# B&R Automation Studio project MIG1
Automation Studio 4.12.7.113 SP; technology packages: Acp10Arnc0 1.0.0

## Configuration X20CP0484

CPU X20CP0484-1, AutomationRuntime E4.53, Build 4.1.2, Vc V4.52.0

### Task classes (Cpu.sw)
```
Cyclic#1 (cycle 1000 us, tolerance 10000 us):
  ESAB <- ESAB.prg
  LincolnPS <- LincolnPS.prg
  UDP_Client <- UDP_Client.prg
  TML_srv <- TML_srv.prg
Cyclic#2 (cycle 4000 us, tolerance 40000 us):
  MainProc <- MainProc.prg
Cyclic#3 (cycle 8000 us, tolerance 48000 us):
  Master <- Master.prg
Cyclic#4 (cycle 100000 us, tolerance 100000 us):
  HMI <- HMI.prg
Cyclic#8 (cycle 10000 us, tolerance 30000000 us):
  Program <- Program.prg [disabled]
  UDP <- UDP.prg [disabled]
  TcpCam <- TcpCam.prg [disabled]
VcDataObjects: Visu <- Visu.dob
Binaries: vcpfgen, vcnet, udbdef, vcrt, vcctext, vctcal, vccslider, Visu03, vcfile, vcgclass, vcpdsw, vccshape, arial, vccbmp, vcmgr, vcchspot, vcdsloc, vcfntttf, Visu02, vccovl, vcshared, arialbd, vcalarm, vcpdvnc, vccbtn, vcbclass, vcdsint, vccpwd, TCData, vccnum, Visu01, vccstr, vccpopup, vccddbox, vccdt, vccline, vcclbox, visvc, verabd, arialbi, vcpkat, vcctrend, iomap, asfw, Role, ashwac, sysconf, ashwd, User, arconfig
Libraries: AsXml, AsUDP, runtime, ETHERNET, standard, dvframe, asstring, AsTCP, AsHydCon, sys_lib, FileUser, FileIO, brsystem, LoopConR, DataObj, AsIOTime, XMLp_Lib, AsMbTCPS, AsMbTCP, vcresman, astime, visapi
```

### Hardware
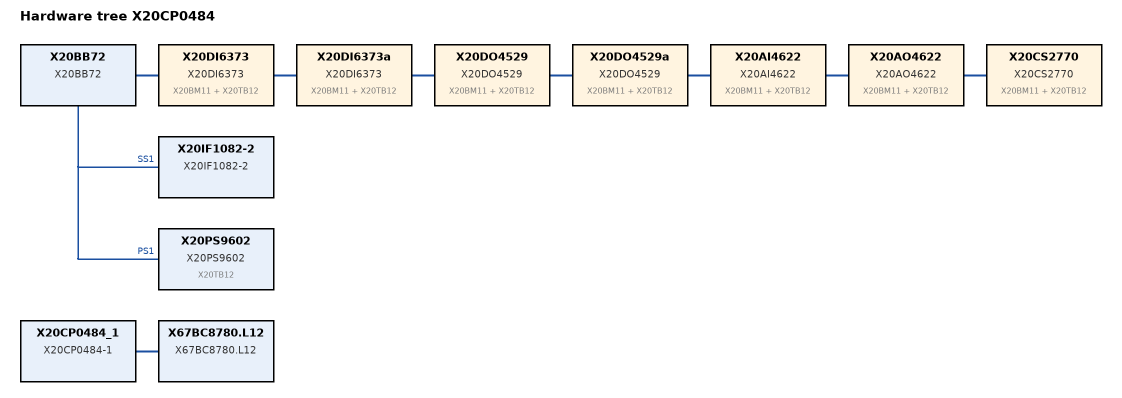
```
X20AI4622 : X20AI4622 v1.0.5.0  [SS1 -> X20TB12a.SS; SL -> X20BM11.SL1]
  Supervision = off
X20AO4622 : X20AO4622 v1.1.0.0  [SS1 -> X20TB12b.SS; SL -> X20BM11a.SL1]
  Supervision = off
X20BB72 : X20BB72 v1.2.0.0
  Connector IF1:
    ActivateIna = 0
  Connector IF6:
    CycleTime = 1000
X20BM11 : X20BM11 v1.1.0.0  [X2X1 -> X20BM11d.X2X2]
X20BM11a : X20BM11 v1.1.0.0  [X2X1 -> X20BM11.X2X2]
X20BM11b : X20BM11 v1.1.0.0  [X2X1 -> X20BB72.IF6]
X20BM11c : X20BM11 v1.1.0.0  [X2X1 -> X20BM11n.X2X2]
X20BM11d : X20BM11 v1.1.0.0  [X2X1 -> X20BM11c.X2X2]
X20BM11m : X20BM11 v1.1.0.0 (Disabled=true)  [X2X1 -> X20BM11a.X2X2]
X20BM11n : X20BM11 v1.1.0.0  [X2X1 -> X20BM11b.X2X2]
X20CP0484_1 : X20CP0484-1 v1.4.0.0
  Connector IF2:
    ActivateDevice = 1
  Connector IF3:
    DNAConfiguration = manual
  ConfigurationID = RemWeld_Config1
  PermanentPvSize = 2048
  RemanentGlobalPvSize = 128
  TimerDeviceType = EPLX2X
  TimerDevice = X20CP0484_1.IF3
  Cyclic1Duration = 1000
  Cyclic1Tolerance = 10000
  Cyclic2Duration = 4000
  Cyclic2Tolerance = 40000
  Cyclic3Duration = 8000
  Cyclic3Tolerance = 48000
  Cyclic4Duration = 100000
  Cyclic4Tolerance = 100000
  Cyclic5Duration = 200000
  Cyclic5Tolerance = 200000
  Cyclic6Duration = 500000
  Cyclic6Tolerance = 500000
  Cyclic7Duration = 1000000
  Cyclic7Tolerance = 1000000
  Cyclic8Duration = 10000
  Cyclic8Tolerance = 30000000
X20CS2770 : X20CS2770 v1.9.1.0 (Disabled=true)  [SS1 -> X20TB12n.SS; SL -> X20BM11m.SL1]
  Connector IF1 (Disabled=true)
  Connector IF2 (Disabled=true)
  Supervision = off
  CANdataFormat01 = UINT
  Baudrate02 = 250000
  CANdataFormat02 = UINT
X20DI6373 : X20DI6373 v1.0.1.0  [SS1 -> X20TB12c.SS; SL -> X20BM11b.SL1]
  Supervision = off
X20DI6373a : X20DI6373 v1.0.1.0  [SS1 -> X20TB12o.SS; SL -> X20BM11n.SL1]
  Supervision = off
X20DO4529 : X20DO4529 v1.2.0.0  [SS1 -> X20TB12d.SS; SL -> X20BM11c.SL1]
  Supervision = off
X20DO4529a : X20DO4529 v1.2.0.0  [SS1 -> X20TB12e.SS; SL -> X20BM11d.SL1]
  Supervision = off
X20IF1082-2 : X20IF1082-2 v1.14.0.0  [SS -> X20BB72.SS1]
  Connector IF1:
    EplNatSubnet = 192.168.102.0
X20PS9602 : X20PS9602 v1.1.0.0  [PS -> X20BB72.PS1; SS1 -> X20TB12.SS]
  Supervision = off
X20TB12 : X20TB12 v1.0.0.0
X20TB12a : X20TB12 v1.0.0.0
X20TB12b : X20TB12 v1.0.0.0
X20TB12c : X20TB12 v1.0.0.0
X20TB12d : X20TB12 v1.0.0.0
X20TB12e : X20TB12 v1.0.0.0
X20TB12n : X20TB12 v1.0.0.0 (Disabled=true)
X20TB12o : X20TB12 v1.0.0.0
X67BC8780.L12 : X67BC8780.L12 v2.14.0.0 (Disabled=true)  [PLK1 -> X20CP0484_1.IF3 [Cable Type=PowerlinkCable, Length=10, Version=1.0.0.3]]
  Connector IF1 (Disabled=true)
```

### Cpu.per - X20CP0484_1/Cpu.per
```iecst
VAR_CONFIG
	permMemInit AT %MX0; (* *)
	TravelSpeed AT %M4; (* *)
	OLD_MTR_POS AT %MD8; (* *)
	CurCalib AT %M72; (* *)
	permMem AT %M468; (* *)
	MachCfg AT %M1620; (* *)
END_VAR
```

### IoMap.iom - X20CP0484_1/IoMap.iom
```iecst
VAR_CONFIG
	::TML_mgr[0].hrdw[0].TXCountReadBack AT %IB."X20CS2770".TX01CountReadBack;
	::TML_mgr[0].hrdw[0].RXDataSize0 AT %IB."X20CS2770".RX01DataSize;
	::TML_mgr[0].hrdw[0].RXIdent0 AT %ID."X20CS2770".RX01Ident;
	::TML_mgr[0].hrdw[0].RXData0Word0[0] AT %IW."X20CS2770".RX01DataWord0;
	::TML_mgr[0].hrdw[0].RXData0Word0[1] AT %IW."X20CS2770".RX01DataWord1;
	::TML_mgr[0].hrdw[0].RXData0Word0[2] AT %IW."X20CS2770".RX01DataWord2;
	::TML_mgr[0].hrdw[0].RXData0Word0[3] AT %IW."X20CS2770".RX01DataWord3;
	::TML_mgr[0].hrdw[0].TXCount AT %QB."X20CS2770".TX01Count;
	::TML_mgr[0].hrdw[0].TXDataSize AT %QB."X20CS2770".TX01DataSize; (*Data length TX object *)
	::TML_mgr[0].hrdw[0].TXIdent AT %QD."X20CS2770".TX01Ident;
	::TML_mgr[0].hrdw[0].TXDataWord0[0] AT %QW."X20CS2770".TX01DataWord0;
	::TML_mgr[0].hrdw[0].TXDataWord0[1] AT %QW."X20CS2770".TX01DataWord1;
	::TML_mgr[0].hrdw[0].TXDataWord0[2] AT %QW."X20CS2770".TX01DataWord2;
	::TML_mgr[0].hrdw[0].TXDataWord0[3] AT %QW."X20CS2770".TX01DataWord3;
	::TML_mgr[0].hrdw[1].RXCount AT %IB."X20CS2770".RX02Count;
	::TML_mgr[0].hrdw[1].TXCountReadBack AT %IB."X20CS2770".TX02CountReadBack;
	::TML_mgr[0].hrdw[1].RXDataSize0 AT %IB."X20CS2770".RX02DataSize;
	::TML_mgr[0].hrdw[1].RXIdent0 AT %ID."X20CS2770".RX02Ident;
	::TML_mgr[0].hrdw[1].RXData0Word0[0] AT %IW."X20CS2770".RX02DataWord0;
	::TML_mgr[0].hrdw[1].RXData0Word0[1] AT %IW."X20CS2770".RX02DataWord1;
	::TML_mgr[0].hrdw[1].RXData0Word0[2] AT %IW."X20CS2770".RX02DataWord2;
	::TML_mgr[0].hrdw[1].RXData0Word0[3] AT %IW."X20CS2770".RX02DataWord3;
	::TML_mgr[0].hrdw[1].TXCount AT %QB."X20CS2770".TX02Count;
	::TML_mgr[0].hrdw[1].TXDataSize AT %QB."X20CS2770".TX02DataSize; (*Data length TX object *)
	::TML_mgr[0].hrdw[1].TXIdent AT %QD."X20CS2770".TX02Ident;
	::TML_mgr[0].hrdw[1].TXDataWord0[0] AT %QW."X20CS2770".TX02DataWord0;
	::TML_mgr[0].hrdw[1].TXDataWord0[1] AT %QW."X20CS2770".TX02DataWord1;
	::TML_mgr[0].hrdw[1].TXDataWord0[2] AT %QW."X20CS2770".TX02DataWord2;
	::TML_mgr[0].hrdw[1].TXDataWord0[3] AT %QW."X20CS2770".TX02DataWord3;
	::Main_IO.Inp[0] AT %IX."X20DI6373".DigitalInput01;
	::VoltCmd_Out AT %QW."X20AO4622".AnalogOutput02;
	::Main_IO.Inp[1] AT %IX."X20DI6373".DigitalInput02;
	::Main_IO.Inp[2] AT %IX."X20DI6373".DigitalInput03;
	::Main_IO.Inp[3] AT %IX."X20DI6373".DigitalInput04;
	::Main_IO.Inp[4] AT %IX."X20DI6373".DigitalInput05;
	::Main_IO.Inp[5] AT %IX."X20DI6373".DigitalInput06;
	::Main_IO.Inp[6] AT %IX."X20DI6373a".DigitalInput01;
	::Main_IO.Inp[7] AT %IX."X20DI6373a".DigitalInput02;
	::Main_IO.Inp[8] AT %IX."X20DI6373a".DigitalInput03;
	::Main_IO.Inp[9] AT %IX."X20DI6373a".DigitalInput04;
	::Main_IO.Inp[10] AT %IX."X20DI6373a".DigitalInput05;
	::Main_IO.Inp[11] AT %IX."X20DI6373a".DigitalInput06;
	::Main_IO.Out[0] AT %QX."X20DO4529".DigitalOutput01;
	::Main_IO.Out[1] AT %QX."X20DO4529".DigitalOutput02;
	::Main_IO.Out[2] AT %QX."X20DO4529".DigitalOutput03;
	::Main_IO.Out[3] AT %QX."X20DO4529".DigitalOutput04;
	::Main_IO.Out[4] AT %QX."X20DO4529a".DigitalOutput01;
	::Main_IO.Out[5] AT %QX."X20DO4529a".DigitalOutput02;
	::Main_IO.Out[6] AT %QX."X20DO4529a".DigitalOutput03;
	::Main_IO.Out[7] AT %QX."X20DO4529a".DigitalOutput04;
END_VAR
```

## Configuration X20CP1585S

CPU X20CP1585, AutomationRuntime J4.93, Build 4.1.2, Safety 1.10, Vc V4.73.2

### Hardware
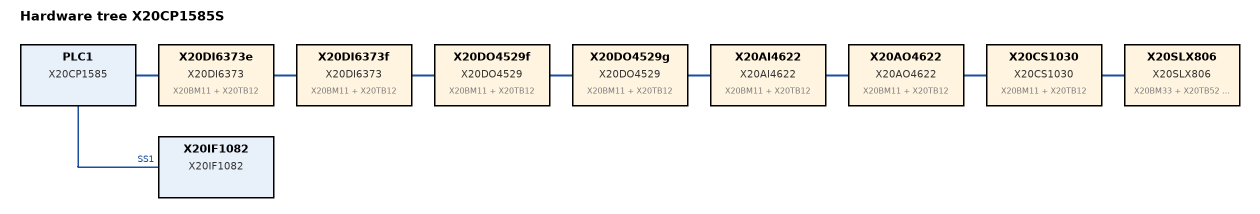
```
PLC1 : X20CP1585 v1.10.0.0
  Connector IF2:
    ActivateDevice = 1
    Mode = Manual
    InternetAddress = 192.168.10.123
    SubnetMask = 255.255.255.0
    Vnc1
    VncVcObjectName1 = Visu
    VncKeyMappingFile1 = VC\PS2-Keyboard.dis
    VncAuthentication1 = 1
    VncPasswordViewControl1 = c
    VncMaxConnections1 = 3
    VncRefreshRate1 = 100
    VncTitle1 = MIG
    Vnc2
    VncVcObjectName2 = Visu1
    VncKeyMappingFile2 = VC\PS2-Keyboard1.dis
    VncAuthentication2 = 1
    VncPasswordViewControl2 = c
    VncPortNumber2 = 5901
    VncRefreshRate2 = 200
  Connector IF3:
    ActivatePowerlink = 0
    DNAConfiguration = manual
    CycleTime = 800
    EplNatSubnet = 192.168.102.0
    HostName = pwl
    InternetAddress = 192.168.11.123
    SubnetMask = 255.255.255.0
    InaNodeNumber = 1
  Connector IF6:
    CycleTime = 800
  ConfigurationID = MIG-26July21
  UserPartitionSize = 256
  UserRamSize = 770048
  PermanentPvSize = 96000
  RemanentGlobalPvSize = 15000
  VolatileGlobalPvSize = 3300000
  TimerDeviceType = EPLX2X
  TimerDevice = PLC1.IF3
  TaskClassIdleTime = 1600
  Cyclic1Duration = 800
  Cyclic1Tolerance = 8000
  Cyclic1Stack = 16000
  Cyclic2Duration = 2400
  Cyclic2Tolerance = 24000
  Cyclic2Stack = 65536
  Cyclic3Duration = 4800
  Cyclic3Tolerance = 24000
  Cyclic4Duration = 24000
  Cyclic4Tolerance = 48000
  Cyclic4Stack = 65536
  Cyclic5Duration = 102400
  Cyclic5Tolerance = 204800
  Cyclic6Duration = 409600
  Cyclic6Tolerance = 409600
  Cyclic7Duration = 20000000
  Cyclic7Tolerance = 20000000
  Cyclic8Duration = 8000
  Cyclic8Tolerance = 40000000
  FileDevice1
  FileDeviceName1 = XML
  FileDevicePath1 = F:\XML
  FileDevice2
  FileDeviceName2 = USB1
  FileDevicePath2 = IF4
  FileDevice3
  FileDeviceName3 = USB2
  FileDevicePath3 = IF5
  FileDevice4
  FileDeviceName4 = REPORTS
  FileDevicePath4 = F:\Reports
  FtpUser1
  FtpUsername1 = anonymous
  FtpUserPassword1 = ilVrWe+rnGADVB+XCj+0qQ/lTsJeu4vW1xfWuH+9Xv8=
  FtpUserSalt1 = NATz6vdL
  FTPAccessRight1 = 0
X20AI4622 : X20AI4622 v1.0.5.0  [SS1 -> X20TB12.SS; SL -> X20BM11.SL1]
  Supervision = off
X20AO4622 : X20AO4622 v1.1.0.0  [SS1 -> X20TB12a.SS; SL -> X20BM11a.SL1]
  Supervision = off
X20BM11 : X20BM11 v1.1.0.0  [X2X1 -> X20BM11p.X2X2]
X20BM11a : X20BM11 v1.1.0.0  [X2X1 -> X20BM11.X2X2]
X20BM11b : X20BM11 v1.1.0.0  [X2X1 -> X20BM11a.X2X2]
X20BM11m : X20BM11 v1.1.0.0  [X2X1 -> PLC1.IF6]
X20BM11n : X20BM11 v1.1.0.0  [X2X1 -> X20BM11m.X2X2]
X20BM11o : X20BM11 v1.1.0.0  [X2X1 -> X20BM11n.X2X2]
X20BM11p : X20BM11 v1.1.0.0  [X2X1 -> X20BM11o.X2X2]
X20BM33 : X20BM33 v1.1.0.0 (Disabled=true)  [X2X1 -> X20BM11b.X2X2]
X20CS1030 : X20CS1030 v1.4.2.0  [SS1 -> X20TB12b.SS; SL -> X20BM11b.SL1]
  Supervision = off
X20DI6373e : X20DI6373 v1.0.1.0  [SS1 -> X20TB12q.SS; SL -> X20BM11m.SL1]
  Supervision = off
X20DI6373f : X20DI6373 v1.0.1.0  [SS1 -> X20TB12r.SS; SL -> X20BM11n.SL1]
  Supervision = off
X20DO4529f : X20DO4529 v1.2.0.0  [SS1 -> X20TB12s.SS; SL -> X20BM11o.SL1]
  Supervision = off
X20DO4529g : X20DO4529 v1.2.0.0  [SS1 -> X20TB12t.SS; SL -> X20BM11p.SL1]
  Supervision = off
X20IF1082 : X20IF1082 v1.6.0.0 (Disabled=true)  [SS -> PLC1.SS1]
  Connector IF1 (Disabled=true)
    ActivatePowerlink = 0
    DNAConfiguration = manual
    InternetAddress = 192.168.1.123
    SubnetMask = 255.255.255.0
X20SLX806 : X20SLX806 v1.10.12.1 (Disabled=true)  [SS1 -> X20TB52.SS; SS2 -> X20TB52a.SS; SL -> X20BM33.SL1]
  Supervision = off
  SafeProject = SafeLOGIC-1
  SafeDesigner = 4.2.5.4
X20TB12 : X20TB12 v1.0.0.0
X20TB12a : X20TB12 v1.0.0.0
X20TB12b : X20TB12 v1.0.0.0
X20TB12q : X20TB12 v1.0.0.0
X20TB12r : X20TB12 v1.0.0.0
X20TB12s : X20TB12 v1.0.0.0
X20TB12t : X20TB12 v1.0.0.0
X20TB52 : X20TB52 v1.0.0.1 (Disabled=true)
X20TB52a : X20TB52 v1.0.0.1 (Disabled=true)
```

- Safety project (password-protected, skipped)

## Configuration X20CP1685S

CPU X20CP1685, AutomationRuntime J4.93, Build 4.1.2, Safety 1.10, Vc V4.73.2

### Hardware
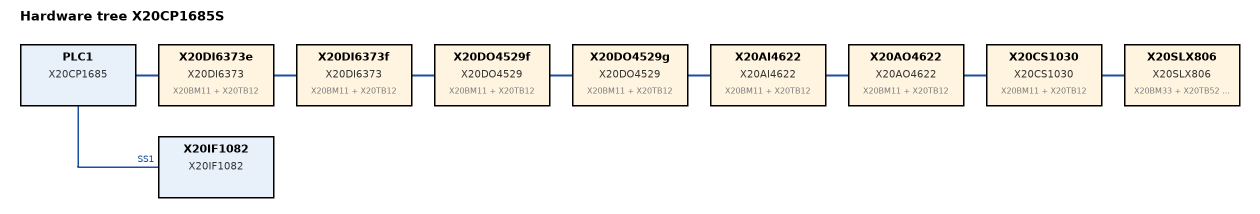
```
PLC1 : X20CP1685 v1.5.0.0
  Connector IF2:
    ActivateDevice = 1
    Mode = Manual
    InternetAddress = 192.168.10.123
    SubnetMask = 255.255.255.0
    Vnc1
    VncVcObjectName1 = Visu
    VncKeyMappingFile1 = VC\PS2-Keyboard.dis
    VncAuthentication1 = 1
    VncPasswordViewControl1 = c
    VncMaxConnections1 = 3
    VncRefreshRate1 = 100
    VncTitle1 = MIG
    Vnc2
    VncVcObjectName2 = Visu1
    VncKeyMappingFile2 = VC\PS2-Keyboard1.dis
    VncAuthentication2 = 1
    VncPasswordViewControl2 = c
    VncPortNumber2 = 5901
    VncRefreshRate2 = 200
  Connector IF3:
    ActivatePowerlink = 0
    DNAConfiguration = manual
    CycleTime = 800
    EplNatSubnet = 192.168.102.0
    HostName = pwl
    InternetAddress = 192.168.11.123
    SubnetMask = 255.255.255.0
    InaNodeNumber = 1
  Connector IF6:
    CycleTime = 800
  ConfigurationID = MIG-26July21
  UserPartitionSize = 256
  UserRamSize = 770048
  PermanentPvSize = 96000
  RemanentGlobalPvSize = 15000
  VolatileGlobalPvSize = 3300000
  TimerDeviceType = EPLX2X
  TimerDevice = PLC1.IF3
  TaskClassIdleTime = 1600
  Cyclic1Duration = 800
  Cyclic1Tolerance = 8000
  Cyclic1Stack = 16000
  Cyclic2Duration = 2400
  Cyclic2Tolerance = 24000
  Cyclic2Stack = 65536
  Cyclic3Duration = 4800
  Cyclic3Tolerance = 24000
  Cyclic4Duration = 24000
  Cyclic4Tolerance = 48000
  Cyclic4Stack = 65536
  Cyclic5Duration = 102400
  Cyclic5Tolerance = 204800
  Cyclic6Duration = 409600
  Cyclic6Tolerance = 409600
  Cyclic7Duration = 20000000
  Cyclic7Tolerance = 20000000
  Cyclic8Duration = 8000
  Cyclic8Tolerance = 40000000
  FileDevice1
  FileDeviceName1 = XML
  FileDevicePath1 = F:\XML
  FileDevice2
  FileDeviceName2 = USB1
  FileDevicePath2 = IF4
  FileDevice3
  FileDeviceName3 = USB2
  FileDevicePath3 = IF5
  FileDevice4
  FileDeviceName4 = REPORTS
  FileDevicePath4 = F:\Reports
  FtpUser1
  FtpUsername1 = anonymous
  FtpUserPassword1 = ilVrWe+rnGADVB+XCj+0qQ/lTsJeu4vW1xfWuH+9Xv8=
  FtpUserSalt1 = NATz6vdL
  FTPAccessRight1 = 0
X20AI4622 : X20AI4622 v1.0.5.0  [SS1 -> X20TB12.SS; SL -> X20BM11.SL1]
  Supervision = off
X20AO4622 : X20AO4622 v1.1.0.0  [SS1 -> X20TB12a.SS; SL -> X20BM11a.SL1]
  Supervision = off
X20BM11 : X20BM11 v1.1.0.0  [X2X1 -> X20BM11p.X2X2]
X20BM11a : X20BM11 v1.1.0.0  [X2X1 -> X20BM11.X2X2]
X20BM11b : X20BM11 v1.1.0.0  [X2X1 -> X20BM11a.X2X2]
X20BM11m : X20BM11 v1.1.0.0  [X2X1 -> PLC1.IF6]
X20BM11n : X20BM11 v1.1.0.0  [X2X1 -> X20BM11m.X2X2]
X20BM11o : X20BM11 v1.1.0.0  [X2X1 -> X20BM11n.X2X2]
X20BM11p : X20BM11 v1.1.0.0  [X2X1 -> X20BM11o.X2X2]
X20BM33 : X20BM33 v1.1.0.0 (Disabled=true)  [X2X1 -> X20BM11b.X2X2]
X20CS1030 : X20CS1030 v1.4.2.0  [SS1 -> X20TB12b.SS; SL -> X20BM11b.SL1]
  Supervision = off
X20DI6373e : X20DI6373 v1.0.1.0  [SS1 -> X20TB12q.SS; SL -> X20BM11m.SL1]
  Supervision = off
X20DI6373f : X20DI6373 v1.0.1.0  [SS1 -> X20TB12r.SS; SL -> X20BM11n.SL1]
  Supervision = off
X20DO4529f : X20DO4529 v1.2.0.0  [SS1 -> X20TB12s.SS; SL -> X20BM11o.SL1]
  Supervision = off
X20DO4529g : X20DO4529 v1.2.0.0  [SS1 -> X20TB12t.SS; SL -> X20BM11p.SL1]
  Supervision = off
X20IF1082 : X20IF1082 v1.6.0.0 (Disabled=true)  [SS -> PLC1.SS1]
  Connector IF1 (Disabled=true)
    ActivatePowerlink = 0
    DNAConfiguration = manual
    InternetAddress = 192.168.1.123
    SubnetMask = 255.255.255.0
X20SLX806 : X20SLX806 v1.10.12.1 (Disabled=true)  [SS1 -> X20TB52.SS; SS2 -> X20TB52a.SS; SL -> X20BM33.SL1]
  Supervision = off
  SafeProject = SafeLOGIC-1
  SafeDesigner = 4.2.5.4
X20TB12 : X20TB12 v1.0.0.0
X20TB12a : X20TB12 v1.0.0.0
X20TB12b : X20TB12 v1.0.0.0
X20TB12q : X20TB12 v1.0.0.0
X20TB12r : X20TB12 v1.0.0.0
X20TB12s : X20TB12 v1.0.0.0
X20TB12t : X20TB12 v1.0.0.0
X20TB52 : X20TB52 v1.0.0.1 (Disabled=true)
X20TB52a : X20TB52 v1.0.0.1 (Disabled=true)
```

### Cpu.per - PLC1/Cpu.per
```iecst
(********************************************************************
 * COPYRIGHT -- wsi
 ********************************************************************
 * File: Cpu.per
 * Author: wsi
 * Created: May 14, 2013
 ********************************************************************
 * Declaration of permanent variables
 ********************************************************************)
VAR_CONFIG
	permMemInit AT %MX0; (* *)
	TravelSpeed AT %M4; (* *)
	OLD_MTR_POS AT %MD8; (* *)
	CurCalib AT %M72; (* *)
	permMem AT %M468; (* *)
	MachCfg AT %M1620; (* *)
END_VAR
```

### IoMap.iom - PLC1/IoMap.iom
```iecst
(********************************************************************
 * COPYRIGHT -- wsi
 ********************************************************************
 * File: IoMap.iom
 * Author: wsi
 * Created: May 14, 2013
 ********************************************************************
 * IO mapping file
 ********************************************************************)
VAR_CONFIG
	::Main_IO.Inp[0] AT %IX."X20DI6373e".DigitalInput01;
	::Main_IO.Inp[1] AT %IX."X20DI6373e".DigitalInput02;
	::Main_IO.Inp[2] AT %IX."X20DI6373e".DigitalInput03;
	::Main_IO.Inp[3] AT %IX."X20DI6373e".DigitalInput04;
	::Main_IO.Inp[4] AT %IX."X20DI6373e".DigitalInput05;
	::Main_IO.Inp[5] AT %IX."X20DI6373e".DigitalInput06;
	::Main_IO.Inp[6] AT %IX."X20DI6373f".DigitalInput01;
	::Main_IO.Inp[7] AT %IX."X20DI6373f".DigitalInput02;
	::Main_IO.Inp[8] AT %IX."X20DI6373f".DigitalInput03;
	::Main_IO.Inp[9] AT %IX."X20DI6373f".DigitalInput04;
	::Main_IO.Inp[10] AT %IX."X20DI6373f".DigitalInput05;
	::Main_IO.Inp[11] AT %IX."X20DI6373f".DigitalInput06;
	::Main_IO.Out[0] AT %QX."X20DO4529f".DigitalOutput01;
	::Main_IO.Out[1] AT %QX."X20DO4529f".DigitalOutput02;
	::Main_IO.Out[2] AT %QX."X20DO4529f".DigitalOutput03;
	::Main_IO.Out[3] AT %QX."X20DO4529f".DigitalOutput04;
	::Main_IO.Out[4] AT %QX."X20DO4529g".DigitalOutput01;
	::Main_IO.Out[5] AT %QX."X20DO4529g".DigitalOutput02;
	::Main_IO.Out[6] AT %QX."X20DO4529g".DigitalOutput03;
	::Main_IO.Out[7] AT %QX."X20DO4529g".DigitalOutput04;
	::VoltCmd_Out AT %QW."X20AO4622".AnalogOutput02;
END_VAR
```

## Logical view

Binary libraries used (declarations not repeated): operator, runtime, astime, AsIecCon, AsUDP, standard, dvframe, asstring, AsTCP, AsHydCon 3.10.0, sys_lib, brsystem, LoopConR 4.10.0, DataObj, AsIOTime, AsMbTCPS, bglibas, AsXml, sprintf2, NcGlobal 3.13.1, Acp10man 3.13.1, Acp10par 3.13.1, AsMbTCP, AsSafety, FileIO, ETHERNET, visapi

### GlobalDef.h
```c
#include <bur/plctypes.h>

#ifndef _GLOBAL_DEF_H
#define _GLOBAL_DEF_H

#ifdef _DEFAULT_INCLUDES
#include <AsDefault.h>
#endif

#include <..\Lib\WSI_types.h>
#include <..\Lib\LoggerLib.h>

#include <..\Lib\arclink\arclink.h>

// "192.168.10.11"   	TML -> CAN conerter
// "192.168.10.2"   	Lincoln Power Supply
// "192.168.10.110"  	VNC - Pendant Screen
// "192.168.10.13" 		My Laptop

//#define SOFTWARE_VERSION    "MIG 09 June 2023V" // two new mode : 169 Carbon & 171 Stainless steel

//#define SOFTWARE_VERSION    "MIG 12 June 2023B" // two new mode : 169 Carbon & 171 Stainless steel

//#define SOFTWARE_VERSION    "MIG 14 June 2023H" // ta dziala przy tescie

//#define SOFTWARE_VERSION    "MIG 20 June 2023F" // FINAL GOOD VERSION req.: MIG 04 Nov 2022 new AHC Rel Move.m

//#define SOFTWARE_VERSION    "MIG 21 June 2023Y" //

//#define SOFTWARE_VERSION    "MIG 22 June 2023H" // Dobrze dziala - sprawdzona z Martin i David

//#define SOFTWARE_VERSION    "MIG 23 June 2023A" // Gas Solenoid in ArcLink

//#define SOFTWARE_VERSION    "MIG 9 Aug 2023C" // Nie dziala - przy stopie bez error WF jechal

//#define SOFTWARE_VERSION    "MIG 9 Aug 2023E"

//#define SOFTWARE_VERSION    "MIG 10 Aug 2023F" // DObra stabilna wersja
//#define SOFTWARE_VERSION    "MIG 11 Aug 2023F" // drobna poprawka w tekscie na ekranie

//#define SOFTWARE_VERSION    "MIG 23 Oct 2024A"  // weld report added

//#define SOFTWARE_VERSION    "MIG5 14 Nov 2024A"  // TVL indexing from trigger

//#define SOFTWARE_VERSION    "MIG 30 Jan 2025F"  // Ramp for amps in gauging , TVL indexing from trigger

//#define SOFTWARE_VERSION    "MIG 08 Aug 2025K"  // Gouging over current protection

//#define SOFTWARE_VERSION    "MIG 14 Aug 2025A"  // No Gouging over current protection & No repeat bead protection when gouging

//#define SOFTWARE_VERSION    "MIG 04 Sept 2025K"  // Report data display
//#define SOFTWARE_VERSION    "MIG 05 Sept 2025K"  // Report data display
#define SOFTWARE_VERSION    "MIG 26 Sept 2025F"  // bypass CheckIndxDone()

//////////////////////////////////////////
#define SERVO_NUM  6 // number of used servo

#define VISIBLE 	0
#define INVISIBLE 	1

#define MAX_PARAM_NUM 96

#define TravelSpeedAO_Indx 				0
#define ArcVoltsAO_Indx  				1
#define	WireFeedSpeedAO_Indx  			2
#define	AHCCurrentSPAO_Indx  			3
#define	AHCToleranceAO_Indx  			4
#define	OSCSpeedAO_Indx  				5

#define	Index_Dist_H_Indx  				6
#define Index_Dist_L_Indx				7

#define	Index_Jog_Speed_Indx  			8
#define	Index_Step_Speed_Indx  			9

#define	TVL_Jog_Speed_Indx  			10
#define WF_Jog_Speed_Indx  				11

#define	Index_PreDlyTime_Indx  			12
#define	Index_PostDlyTime_Indx  		13

////
#define	OSC_AmplitAO_Indx  				14
#define	OSC_DwellInAO_Indx  			15
#define	OSC_DwellOutAO_Indx  			16
#define	OSC_JogSpeedAO_Indx  			17
#define	OSC_StepDistAO_Indx  			18

/////
#define	AHC_JogSpeedAO_Indx  			19
#define AHC_Response_Indx  				20
#define AHC_Integrator_Indx  			21

////////////
#define TVL_Calibr_Vel_Low				25
#define TVL_Calibr_Vel_High				26
#define TVL_Calibr_Dist					27
////////////
#define WF_Calibr_Vel_Low				30
#define WF_Calibr_Vel_High				31
#define WF_Calibr_Time					32

/////// Ramps
#define TVL_Ramp						50
#define TVL_Return_Speed				51

#define WF_Ramp							52
#define TVL_Skip_Speed					53

////  GAS

#define GAS_PrePurge					54
#define GAS_PostPurge					55

////  Weld Mode

#define StanBy_Time						56
#define Weld_Pinch						57
#define Weld_Trim						58
#define Weld_UltimArc					59

#define AMPS_Calibr_Low					60
#define AMPS_Calibr_High				61

#define BURN_BACK_Tm					62

#define WF_SlowSpeed					63

#define AHC_Retrack_Dist  				64

#define GOUG_Volts  				    65
#define GOUG_Amps 				    	66

#define ARC_Start_Tmo					67
#define ARC_NotActive_Level				68

#define OSC_OFF_Tm						69

#define GOUG_Amps_Init 				    70
#define GOUG_Amps_Ramp 				    71

#define GOUG_Amps_Limit 				72
#define GOUG_Amps_Limit_Tm 				73

#define Wire_Dim 						74

#define	LastPermMem_Indx  				75

/////////////////////////////////////////////////
#define CALIBR_WF_Indx					0
#define CALIBR_AMPS_Indx				1
#define CALIBR_TVL_Indx					2

///////////////////////
#define WF_Calibr_Indx			0   // speed
#define AMPS_Calibr_Indx		1   // Amp feedback
#define TVL_Calibr_Indx			2   // speed

#define Index_Calibr_Indx		3   // distance
#define OSC_Calibr_Indx			4	// distance
#define ArcVolts_Calibr_Indx	5   // Volts to Power Supply

///////////////////////////
#define mm2inch 0.03936996
#define in_min_2_mm_s 25.4/60.0
#define in_2_mm 25.4

/////////   IO mapping
// Inputs

#define ESTOP_status 5

#define STOP_RST_BTN_LOC 6
#define STOP_RST_BTN 7

#define JOG1_BTN 9
#define JOG2_BTN 10

#define RESET_BTN_LOC 11

//outputs
#define ENABLE_out 3
#define RESET_ESR_Btn_out 4

typedef struct HEAD_typ
{
	plcbit Remote_SW;
	plcbit LocalJog_FWD;
	plcbit LocalJog_REV;

} HEAD_typ;

/////////////////////

typedef struct Mach_Config_typ
{	SINT OSCon;
	SINT IndxDir;
	SINT Indxon;
	SINT IndxExt;
	SINT AHC_Auto;
	SINT WeldMode;
	SINT Weld;
	UINT Weld_mode;
	SINT TorchLastPos;
	SINT TestMode;
	SINT TorchIdleDeg;
	SINT ContinSingle;
	SINT GougingON;
	SINT AHC_BackStep;
	SINT GougHighJogSpeed;
	SINT STOP_TVL_After_SKIP;
	SINT TrigStep_INDX_TVL;
	SINT GougAutAHC;
	SINT spare[13];

} Mach_Config_typ;

typedef struct Analog_Out_Mem_typ
{	float Value;
	float H_Incr;
	float L_Incr;
} Analog_Out_Mem_typ;

typedef struct PermMem_typ
{
	//float TVL_Lo_Limit;
	//float TVL_Hi_Limit;
	struct Analog_Out_Mem_typ Analog_Out[MAX_PARAM_NUM];
} PermMem_typ;

//////////////
typedef struct RS_Channel_typ{
	USINT Status;
	USINT Data[32];
	UINT Len;
	UINT _len_prev;
	UDINT Cntr;
	UDINT Trash_Cntr;
	UINT Msg_ID;
	UINT Msg_Error;

}RS_Channel_typ;

typedef struct EditBox_typ
{	plcbit H_Incr_Plus_Btn;
	plcbit L_Incr_Plus_Btn;
	plcbit H_Incr_Minus_Btn;
	plcbit L_Incr_Minus_Btn;
	plcbit Return_Btn;

	USINT Cmd;

} EditBox_typ;

typedef struct Analog_Out_Module_typ{
	plcstring Name[81];
	float Min_Val;
	float Max_Val;
	//LCRLimScal_typ LimScale;

}Analog_Out_Module_typ;

////  FOR TML Configuration

#define VECTORS_NUM		6
#define TML_SERVO_NUM 	16
#define TML_MGR_NUM 	2

#define TML_AX_TVL 			0
#define TML_AX_OSC 			1
#define TML_AX_AHC 			2
#define TML_AX_WF			3
#define TML_AX_INDX 		4
#define TML_AX_INDX_EXT		5

#define VECT_AX_TVL 		0
#define VECT_AX_OSC 		1
#define VECT_AX_AHC 		2
#define VECT_AX_WF			3
#define VECT_AX_INDX 		4
#define VECT_AX_INDX_EXT	5

////////////////////////////////

// NEW ADDED is below

////////////////////////////////

#define mm2inch 0.03936996
#define in_min_2_mm_s 25.4/60.0
#define in_2_mm 25.4

/*******************************/

#define MODE_NONE 	0
#define MODE_TVL 	1
#define MODE_OSC 	2
#define MODE_AHC 	3
#define MODE_WF 	4
#define MODE_INDX 	5
#define MODE_INDX_EXT 	6

/*******************************/
/*         ALARMS  			****/
/*******************************/

// Alarms Class
#define ERROR_SETUP 		-2
#define ERROR_FATAL 		-1
#define ERROR_MOTOR  		1
#define ERROR_MOTOR_INIT  	2
#define ERROR_TIG_PROC  	3
#define ERROR_COOL_GAS  	4
#define ERROR_TVL  			5
#define ERROR_PENDANT  		6
#define ERROR_ESTOP  		10

// Alarms items
#define ERROR_NONE 0

#define ERROR_DRV_01 1
#define ERROR_DRV_11 11
#define ERROR_DRV_21 21
#define ERROR_DRV_31 31
#define ERROR_DRV_41 41

// Warnings
#define WARN_AVC_LIMITS  0
#define WARN_OSC_LIMITS  1

////   Moved from GlobalTyp.h (ST)

typedef enum Jog_Direction
{	Stop = 0,
	Forward = 1,
	Reverse = 2
} Jog_Direction;

typedef struct ReversingRelay
{	enum Jog_Direction IN;
	//plcbit OUT[4];
	//plcbit Forward;
	//plcbit Reverse;
	//plcbit Stop;
} ReversingRelay;

typedef struct Sequence
{	plcbit _start;
	plcbit _stop;
	plcbit Start_in;
	plcbit Stop_in;
	plcbit Start_out;
	plcbit Stop_out;
	struct TOF startTimer;
	struct TOF stopTimer;
	unsigned short State;
} Sequence;

typedef struct Indexer_typ
{	plcbit Run;
	plcbit Limit_Forward;
	plcbit Limit_Reverse;
	plcbit Direction;
	plcbit Sequence;
	plcbit Start;
	signed char ManualStep;
	float* Speed_Forward;
	float* Speed_Reverse;
	float* Speed_Jog;
	signed short Speed;
	unsigned char state;
	float* Reverse_time;
	float* Forward_time;
	float* PreDly_time;
	float* PostDly_time;
	struct TON timer;
	unsigned short period;
} Indexer_typ;

typedef struct IO_typ{

	plcbit Inp[12];

	plcbit Out[12];

}IO_typ;

/////////////////////////////////////////////////////////////
//////////////////////////////////////////////////////////

typedef struct ESAB_CMD_typ{

plcbit WeldON;
plcbit QuickStop;

plcbit WF_Jog_FWD;
plcbit WF_Jog_REV;

plcbit JogHighSpeed;

plcbit InputArea;

plcbit UpdateParam;

}ESAB_CMD_typ;

typedef struct ESAB_Fbk_typ{

	UINT HeartBeat;

	USINT  Status;
	USINT  StatusMSB;
	plcbit ReadyToStart;
	plcbit Error;
	plcbit InputAreaActive;

	USINT SetRegulType;

	float SetVoltage;
	float SetAmps;
	float SetWF;
	float SetTVL;
	float Req_WF_Speed;
	float Req_TVL_Speed;

	float actVolts;
	float actAmps;
	float actHeat;
	float actWF;

	USINT ErrorNum;
	UINT ErrorCode;
	USINT ErrorSubCode;
	USINT ErrorNodeID;

	USINT NewErrorCode;

}ESAB_Fbk_typ;

typedef struct ESAB_Param_typ{

	float Voltage;
	float Amps;
	USINT RegulType;

}ESAB_Param_typ;

typedef struct ESAB_Msc_typ{

	USINT 	_recev_counts;
	USINT 	_sent_counts;

	plcbit _weldON;
	plcbit _quickStop;

	plcbit _inputArea;

	float _voltage;
	float _amps;
	USINT _regulType;

	plcbit _wF_Jog_FWD;
	plcbit _wF_Jog_REV;

	plcbit _jogHighSpeed;

	USINT _heartBeat;

	USINT _errorNum;

	TON_typ Main_Tmr;
	TON_typ Cmd_Hrbt_Tmr;

}ESAB_Msc_typ;

typedef struct ESAB_typ{
	USINT step;

	ESAB_CMD_typ Cmd;
	ESAB_Param_typ Param;
	ESAB_Fbk_typ Fbk;
	ESAB_Msc_typ Msc;

}ESAB_typ;

///////////////////////////////////////////////////
#endif
```

### GlobalDecl.h
```c
#ifndef _GLOBAL_DECL_H
#define _GLOBAL_DECL_H

#include <bur/plctypes.h>

#include <..\GlobalDef.h>

//#include <..\Lib\arclink\Robot.h>

// For TML comunnication over Ethernet
_GLOBAL RS_Channel_typ TML_Msg_Chan[2] , TML_Data_Chan[2] , UDP_Connect_Send[2];
_GLOBAL USINT Kick_TML_Cmd;
_GLOBAL Arc_Link_typ ArcLink;

_GLOBAL ESAB_typ ESAB_PS;

_GLOBAL plcbit UDP_Ready ,UDP_Restart;

//////////////

_GLOBAL_RETAIN Mach_Config_typ MachCfg;

_GLOBAL plcbit Purge;
_GLOBAL plcbit OSCJog;
_GLOBAL plcbit OSCToggle;
_GLOBAL plcbit GAS_Cmd;
_GLOBAL SINT INDX_Step_Cmd;
_GLOBAL SINT TVL_Step_Cmd;
_GLOBAL plcbit SKIP_Weld_Cmd;
_GLOBAL_RETAIN struct ReversingRelay TravelSpeed;
_GLOBAL struct ReversingRelay TravelJog;
_GLOBAL struct Sequence Seq;
_GLOBAL struct ReversingRelay IndexJog;
_GLOBAL struct ReversingRelay IndexExtJog;
_GLOBAL struct ReversingRelay AHCJog;
_GLOBAL struct ReversingRelay WFJog;
_GLOBAL plcbit pelcoMsgReady;
_GLOBAL unsigned char pelcoPreset;
_GLOBAL unsigned char pelcoCommand;
_GLOBAL unsigned char _pelcoCommand;
_GLOBAL unsigned char pelcoAddress;
_GLOBAL float Slider;
_GLOBAL unsigned char RockerButton;
_GLOBAL unsigned char ToggleSwitch;
_GLOBAL plcbit X20ModuleOK[14];
_GLOBAL plcbit X67ModuleOK[3];
_GLOBAL unsigned short ModulesOK;
_GLOBAL plcbit ESTOP;
_GLOBAL unsigned short visESTOP;
_GLOBAL unsigned char visPage;
_GLOBAL unsigned char visChangePage;
_GLOBAL unsigned short visMaint;
_GLOBAL plcbit SequenceRun_Out;
_GLOBAL plcbit SequenceRun_WF;
_GLOBAL plcbit SequenceRun_OSC;
_GLOBAL plcbit computerPower[2];
_GLOBAL float visTravelSpeed;
_GLOBAL unsigned char cameraCommand;
_GLOBAL_RETAIN plcbit permMemInit;
_GLOBAL unsigned char ledLevel;
_GLOBAL unsigned char cameraPicked;
_GLOBAL plcbit cameraPower;
_GLOBAL float _TravelSpeed;
_GLOBAL unsigned short DisplayInfo;
_GLOBAL plcstring SoftwareVersion[81];
_GLOBAL plcbit MoveEnable;
_GLOBAL USINT LocalJogMode;
_GLOBAL plcbit MachActive;
_GLOBAL TouchAction   Screen_touch;
_GLOBAL plcbit ErrorFromMaster_flag;

// From Head

_GLOBAL HEAD_typ Head;

//  For Files saving

_GLOBAL  SM_obj Screen_sm;
_GLOBAL  SCREEN_obj Screen;
_GLOBAL  FILEMGR_obj FileMgr;
_GLOBAL  FILEOUT_IF File_out;
_GLOBAL  FILEIN_IF File_in;
_GLOBAL XML_Method_typ XMLFile;
_GLOBAL_RETAIN unsigned char ROM_USB;
_GLOBAL_RETAIN plcstring RecipeName[81];

/////////////////////////////////////////////////////
/// For HMI only
_GLOBAL plcbit SetDefault;
_GLOBAL plcbit SetDefault_TVL_Calibr;
_GLOBAL plcbit SetDefault_WF_Calibr;
_GLOBAL plcbit SetDefault_AMPS_Calibr;
_GLOBAL UINT Page_Step;

_GLOBAL UINT PageBtnPress[16];
_GLOBAL UINT EditBox_Vis;
_GLOBAL UINT EditBox_Indx;
_GLOBAL UINT Inc_Plus_Btn_Vis;
_GLOBAL UINT Inc_Minus_Btn_Vis;
_GLOBAL UINT Fwd_Limit_Vis, Rev_Limit_Vis;

_GLOBAL UINT EndOfBead_Stop;
_GLOBAL UINT Sequence_Halt_Cmd;

_GLOBAL UINT AccessLevel;

_GLOBAL plcbit HardwInit_Done;

_GLOBAL Analog_Out_Module_typ Analog_Out_Mod[MAX_PARAM_NUM];
_GLOBAL_RETAIN struct PermMem_typ permMem;
_GLOBAL_RETAIN struct CurCalib_typ CurCalib;
_GLOBAL_RETAIN DINT OLD_MTR_POS[TML_SERVO_NUM];

_GLOBAL UINT NewPageReq_Cmd;
_GLOBAL EditBox_typ EditBox;

_GLOBAL USINT Travel_JOG_Step;

_GLOBAL USINT Travel_JOG_Step_FWD_Cmd , Travel_JOG_Step_REV_Cmd;

_GLOBAL USINT INDX_Limit_Bypass_Btn;

_GLOBAL plcbit LED_One_Blink_Req;

////////////////////////////////////////////
////  For Calibration
_GLOBAL plcstring HMI_Calibr_Intruct_TXT[128];
_GLOBAL UINT HMI_Calibr_Indx;
_GLOBAL USINT HMI_Calibr_Start_Stop , HMI_Calibr_New_User_Input;
_GLOBAL USINT HMI_Calibr_Type_Select;
_GLOBAL USINT HMI_Calibr_NewStart_Btn , HMI_Calibr_Verify_Btn , HMI_Calibr_Resume_Btn;
_GLOBAL USINT HMI_Calibr_Step;
_GLOBAL UINT HMI_Calibr_StartBtn_vis , HMI_Calibr_StopBtn_vis ;//, HMI_Calibr_New_User_Input_vis  ;
_GLOBAL UINT HMI_Calibr_Slop0_vis , HMI_Calibr_Slop1_vis;
_GLOBAL UINT HMI_Calibr_CalculateBtn_vis , HMI_Calibr_SaveBtn_vis , HMI_Calibr_User_Input_vis;
_GLOBAL UINT HMI_Calibr_UserInput_Lock;
_GLOBAL UINT HMI_Calibr_Resume_Btn_vis;
_GLOBAL UINT HMI_Calibr_Step_Done[8];
_GLOBAL UINT HMI_Step_Color[16];
_GLOBAL UINT HMI_Step_Vis[16];
_GLOBAL float HMI_Calibr_Meas_Value;
_GLOBAL Calib_Param_typ TempCalibr;
_GLOBAL float HMI_Calibr_User_Inputs[8];
_GLOBAL float HMI_Calibr_Correct, HMI_Calibr_Error;
_GLOBAL float HMI_Calibr_Slop , HMI_Calibr_Bias;
_GLOBAL float HMI_Calibr_Slop2 , HMI_Calibr_Bias2;

_GLOBAL UINT HMI_AXIS_Disable[6];

_GLOBAL UINT HoldThisAxError;

_GLOBAL float Calibr_Error[8];
_GLOBAL UINT HMI_Calibr_What_vis[8];

// TVL
_GLOBAL float TVL_Calibr_Speed;
_GLOBAL float TVL_Calibr_Distance;
_GLOBAL float TVL_Act_Pos;
_GLOBAL USINT TVL_Start_Err;
_GLOBAL USINT ESAB_Tmo_Err;
_GLOBAL float TVL_Last_Pos;
_GLOBAL Jog_Direction TVL_Last_Dir;

// INDX
_GLOBAL float INDX_Act_Pos;
_GLOBAL float INDX_Home_Pos;
_GLOBAL plcbit INDX_SetHome_Btn;
_GLOBAL float INDX_Last_Pos;

_GLOBAL plcbit WatchIndx;
_GLOBAL UINT ProcError_vis;
_GLOBAL UINT ProcError_Indx;

// AHC
_GLOBAL plcbit AHC_SetHome_Btn;
_GLOBAL float AHC_Scaled_Pos;
_GLOBAL float AHC_MaxPos;
_GLOBAL float AHC_StartPos;
_GLOBAL float AHC_Scaled_MaxPos;
_GLOBAL float AHC_Scaled_StartPos;
_GLOBAL float AHC_Scaled_Fact;

_GLOBAL plcbit ObserveAHC_MaxPos;

// WF
//_GLOBAL SINT  WF_Calibr_Cmd;
_GLOBAL float WF_Calibr_Speed;
_GLOBAL float WF_Calibr_Distance;

_GLOBAL float AMPS_Calibr_Val;

/////////////

_GLOBAL IO_typ Main_IO;
_GLOBAL plcbit ENABLE_sign;
_GLOBAL plcbit STANDBY_sign;

_GLOBAL plcbit RESET_ESR_Btn; // HMI
_GLOBAL UINT RESET_ESR_Btn_vis;

_GLOBAL plcbit Robot_Cmd_RUN , Robot_Cmd_RUN1;

_GLOBAL plcbit HardRestart_Mode;

////////////////////////////////////////////

_GLOBAL SINT OSCJog_Cmd;
///  new
_GLOBAL ERROR_Mgr_typ ErrorMgr;

_GLOBAL plcbit HardwReady;
_GLOBAL plcbit ReadyToOperate;

_GLOBAL UINT HardInit_Step;

_GLOBAL LOGMGR_obj	LogMgr ;
_GLOBAL UDINT LogID; // _VAR_RETAIN;
_GLOBAL StateVectorProxy_typ VectorStateMach[VECTORS_NUM];
_GLOBAL TML_MGR_typ TML_mgr[TML_MGR_NUM];
_GLOBAL TML_typ TML_MTR_INST[TML_SERVO_NUM] ;
_GLOBAL TML_Axis_typ AxisCh[TML_SERVO_NUM];
_GLOBAL float Glbl_TML_CMD_Delay;

_GLOBAL BOOL TML_MTR_CUT_POWER , TML_STOP_SEND_ERROR;
_GLOBAL BOOL KK_HoldEnable;
_GLOBAL plcbit StopStateMachineEvaluation;

_GLOBAL plcbit ResetErrorInTML;

_GLOBAL UINT TVL_Step;
_GLOBAL UINT OSC_Step;
_GLOBAL UINT INDX_Step;
_GLOBAL UINT AHC_Step;
_GLOBAL UINT WF_Step;

_GLOBAL float OSC_Steer;

_GLOBAL plcbit WeldCalibr_Mode;

_GLOBAL TON_typ GAS_ON_Tmr , GAS_OFF_Tmr;
_GLOBAL UINT LED_CMD;

_GLOBAL AzzMovAvgFlt_typ  ActCurrent_Filter;
_GLOBAL float ActCurrrentFbk;
_GLOBAL float ActCurrrentFbk_Calib[2];
_GLOBAL float HMI_Act_Amps;
//_GLOBAL float AHCResponde_Calib[2];
_GLOBAL USINT AHC_Mode;
_GLOBAL float AHC_Move_Target;
_GLOBAL plcbit  AHC_Move_Cmd;

_GLOBAL INT VoltCmd_Out , AmpsCmd_Out;

_GLOBAL AzzRamp_typ AHC_Ramp;
_GLOBAL AzzRamp_typ TVL_Jog_Ramp , INDX_Jog_Ramp , WF_Volt_Ramp , OSC_Jog_Ramp , WF_Run_Ramp ;
_GLOBAL AzzSlimPID_typ AHC_PID;
_GLOBAL azzslimpid_par_typ AHC_PIDParameters;
_GLOBAL plcstring HMI_Error_Txt[32];

_GLOBAL AzzRamp_typ ESAB_Amp_Ramp;

// Just for compatibilty with UniverslCntroller TML_Server
_GLOBAL FILE_RW_typ File_RW; // Dummy structure - do not use
_GLOBAL float ABS_TVL_Pos;
_GLOBAL plcbit ProjectConfig_Hrdw_ERROR;
_GLOBAL plcbit KK_DoNotChangeTMLProgram; // Must be 1
_GLOBAL plcbit KK_TML_PowerON ;

_GLOBAL USINT KK_TVL_Test_step;

_GLOBAL plcstring ErrorMgr_Txt[SERVO_NUM][64];
_GLOBAL plcstring DriveVer_Txt[SERVO_NUM][64];

#endif
```

### Package Logical/Libraries - Global libraries

### Library Logical/Libraries/FileUser (ANSIC, version 0.00.0)
Depends on: sys_lib, FileIO

#### FileUser.fun
```iecst
FUNCTION FU_init : DINT
	VAR_INPUT
		fm_adr : UDINT;
		sDevice : STRING[20];
		Path : STRING[80];
		data_adr : UDINT;
		size : UDINT;
		Type : USINT;
		_if_in_adr : UDINT;
		_if_out_adr : UDINT;
		sDevice2 : STRING[20];
		_fname_adr : UDINT;
		_ftp_adr : UDINT;
		MaxFiles : UINT;
	END_VAR
END_FUNCTION

FUNCTION FU_serv : DINT
	VAR_INPUT
		fm_adr : UDINT;
	END_VAR
END_FUNCTION

FUNCTION FU_setBufPointer : BOOL (*TODO: Add your comment here*)
	VAR_INPUT
		fm_adr : UDINT;
		pMem : UDINT;
		size : UDINT;
	END_VAR
END_FUNCTION
```

#### FileUser.typ
```iecst
TYPE
	FILE_EXT : 	STRUCT
		Name : STRING[4];
	END_STRUCT;
	FILEOUT_IF : 	STRUCT
		OpenDirectory : BOOL;
		OpenFile : UINT;
		CopyFile : BOOL;
		DeleteFile : BOOL;
		PageUp : BOOL;
		SaveAs : BOOL;
		Save : BOOL;
		PageDown : BOOL;
		Refresh : BOOL;
		ClearStatus : BOOL;
		SelectedFileNum : UINT;
		SelectedFile : STRING[34];
		SelectedDirectory : STRING[34];
		NewFileNameBase : STRING[30];
		NewFileName : STRING[34];
		FileSize : UDINT;
		ExtensionIndex : USINT;
		Extension : ARRAY[0..4] OF FILE_EXT;
		StreamEnable : USINT;
		StreamGo : USINT;
		StreamClose : USINT;
		StreamOffset : USINT;
		StreamLength : USINT;
		Stream_adr : USINT;
		pDestDev : STRING[20];
	END_STRUCT;
	FILEMGR_obj : 	STRUCT
		Message : STRING[50];
		Error : USINT;
		Device : STRING[20];
		Path : STRING[80];
		Status : SINT;
		FileLength : UDINT;
		OpenFileName : STRING[35];
		OpenFileNum : USINT;
		OpenFileDate : DATE_AND_TIME;
		Type : UINT;
		BufferSize : UDINT;
		Data_adr : UDINT;
		MaxDirectoryFiles : UINT;
		_if_in_adr : UDINT;
		_if_out_adr : UDINT;
		_fname_adr : UDINT;
		_ftp_adr : UDINT;
		_state : UINT;
		_error : UINT;
		_fileptr : UDINT;
		_numfiles : UDINT;
		_infostatus : UINT;
		_readstatus : UINT;
		_fileopenstatus : UINT;
		_filereadstatus : UINT;
		_filecreatestatus : UINT;
		_filewritestatus : UINT;
		_userfileptr : UINT;
		_dirinfo : DirInfo;
		_dirread : DirRead;
		_fileopen : FileOpen;
		_fileread : FileRead;
		_filedelete : FileDelete;
		_filecopy : FileCopy;
		_filecreate : FileCreate;
		_filewrite : FileWrite;
		_fileclose : FileClose;
	END_STRUCT;
	FILEIN_IF : 	STRUCT
		TotalPageFileNum : UINT;
		TotalDirectoryFileNum : UINT;
		FileNames : ARRAY[0..19] OF STRING[34];
		FileDates : ARRAY[0..19] OF DATE_AND_TIME;
		FileSizes : ARRAY[0..19] OF UDINT;
		OpenFileName : STRING[34];
		PageNum : USINT;
		ExtensionIndex : USINT;
		Status : SINT;
		FileLength : UDINT;
		BufferSize : UDINT;
		StreamReady : BOOL;
		StreamError : BOOL;
		Message : STRING[49];
	END_STRUCT;
END_TYPE
```

#### FileUser.var
```iecst
VAR CONSTANT
	fuFILE_LOAD_OK : SINT := 4;
	fuDRIVE_FILEIO : USINT := 0;
	fuDRIVE_FTP : USINT := 1;
END_VAR
```

#### FileUserSource.c
```c
/********************************************************************
 * COPYRIGHT -- Lenovo
 ********************************************************************
 * Library: FileUser
 * File: FileUserSource.c
 * Author: Frys Electronic
 * Created: September 02, 2009
 * Mofified: 21 Oct 09 - by KK
 *******************************************************************/

#include <bur/plctypes.h>
#include "FileUser.h"
#include <string.h>

/*User Private Library Error Numbers (value assigned as suggested in the B&R help file)*/
#define USER_ERROR_MIN 0xC350
#define USER_ERROR_MAX 0xEA5F
#define USER_ERROR_COB	USER_ERROR_MIN
#define FU_MAX_PAGE_FILES	10
#define FU_MAX_EXT			5
#define FU_DRIVE_FILEIO		0
#define FU_DRIVE_FTP		1
#define FU_DRIVE_STREAM	2

/* Prototypes */
DINT GetExtType( FILEIN_IF *in, FILEOUT_IF *out );
void ConvertToUpper( STRING s[35] );

unsigned short SortDirectory(unsigned long fm_adr);
signed long FU_AddExt(struct FILEOUT_IF* out, struct FILEIN_IF* in);
signed long CreateNewFileName(struct FILEOUT_IF* out);
signed long FindString(plcstring* s, plcstring* ext);

/* LOCAL */
DINT FU_init( 	UDINT fm_adr,  plcstring* sDevice, plcstring* Path, UDINT data_adr, UDINT size, USINT Type, UDINT _if_in_adr, UDINT _if_out_adr,
				plcstring* sDevice2, UDINT _fname_adr, UDINT _ftp_adr, UINT MaxFiles )
{
FILEMGR_obj *fm = ( FILEMGR_obj *) fm_adr;
FILEIN_IF *in;

	/* Default: */
	fm->_state 			= 0;

	fm->_if_in_adr		= _if_in_adr;
	fm->_if_out_adr		= _if_out_adr;
	fm->_fname_adr		= _fname_adr;
	fm->_ftp_adr			= _ftp_adr;
	fm->Type			= Type;
	fm->BufferSize		= size;
	fm->MaxDirectoryFiles	= MaxFiles;
	fm->Data_adr		= data_adr;

	/* */
	strcpy( fm->Device, sDevice );

	/* New Stuff */
	in 					= (FILEIN_IF   *) fm->_if_in_adr;
	in->BufferSize		= fm->BufferSize;

	/* */
	strcpy( fm->Device, sDevice );

	/* Init: DirInfo */
	fm->_dirinfo.enable 	= 1;
	fm->_dirinfo.pDevice	= (UDINT) fm->Device;
	fm->_dirinfo.pPath 		= (UDINT)Path;

	/* Init: DirRead */
	fm->_dirread.enable 	= 1;
	fm->_dirread.pDevice	= (UDINT) fm->Device;
	fm->_dirread.pPath 		= (UDINT)Path;
	fm->_dirread.option 	= FILE_FILE;
	fm->_dirread.data_len 	= sizeof(fiDIR_READ_DATA);

	/* Init: FileOpen */
	fm->_fileopen.enable 	= 1;
	fm->_fileopen.pDevice 	= (UDINT) fm->Device;
	fm->_fileopen.mode 		= FILE_RW;

	/* Init: FileRead */
	fm->_fileread.enable	= 1;
	fm->_fileread.offset 	= 0;
	fm->_fileread.pDest 	= data_adr;
	if ( fm->Type != FU_DRIVE_STREAM )
		fm->_fileread.len 	= fm->BufferSize;

	/* Init: FileDelete */
	fm->_filedelete.enable 	= 1;
	fm->_filedelete.pDevice	= (UDINT) fm->Device;
	fm->_filedelete.pName	= 0;

	/* Init: FileCopy */
	fm->_filecopy.enable	= 1;
	fm->_filecopy.pSrcDev	= (UDINT) fm->Device;
	fm->_filecopy.option	= FILE_OW_DETMEM;
	fm->_filecopy.pDestDev	= (UDINT) sDevice2;

	/* Init: FileCreate */
	fm->_filecreate.enable 	= 1;
	fm->_filecreate.pDevice = (UDINT) fm->Device;

	/* Init: FileWrite */
	fm->_filewrite.enable	= 1;
	fm->_filewrite.offset 	= 0;
	fm->_filewrite.pSrc 	= data_adr;
	if ( fm->Type != FU_DRIVE_STREAM )
		fm->_filewrite.len 	= fm->BufferSize;

	/* Init: FileClose */
	fm->_fileclose.enable	= 1;
	fm->_fileclose.ident 	= 0;

   	return 0;
}
/* Set Buffer Pointer*/
plcbit FU_setBufPointer(unsigned long fm_adr , unsigned long pMem, unsigned long size)
{
FILEMGR_obj *fm			= (FILEMGR_obj *) fm_adr;

	fm->Data_adr		= pMem;
	fm->_filewrite.pSrc = fm->Data_adr;
	fm->_fileread.pDest = fm->Data_adr;

	fm->BufferSize		= size;
	fm->_fileread.len 	= fm->BufferSize;
	fm->_filewrite.len 	= fm->BufferSize;

	return 1;

}

/* Special: Allow Index 0 and 1 */
DINT FU_serv( UDINT fm_adr )
{
FILEMGR_obj *fm			= (FILEMGR_obj *) fm_adr;
FILEIN_IF *in 			= (FILEIN_IF   *) fm->_if_in_adr;
FILEOUT_IF *out			= (FILEOUT_IF  *) fm->_if_out_adr;
fiDIR_READ_DATA *fname;
UINT i,j,StartIndex;
BOOL FilterExt = 0, FileFound = 0;

	/* Open Directory and Delete File does not require data buffer*/
	if((!fm->Data_adr) && (out->OpenFile || out->Save || out->SaveAs)) return -100;

	/* Method: Open Directory */
	switch ( fm->_state )
	{

		/**** Return Directory Information ****/
		case 0:

			if ( out->OpenDirectory ) {

				/* FTP */
				if ( fm->Type == FU_DRIVE_FTP ) {

				}

				/* File IO */
				else {
					/* Reset Status */
					fm->Status = 0;
					/* Reset when Directory Opened */
					in->PageNum	= 0;

					ERRxwarning(0xC351, 1, "FileIO: Open Dir");

					/* Attach Path */
					fm->_dirinfo.pPath		= (UDINT) out->SelectedDirectory;

					/* Call FBK */
					DirInfo(&fm->_dirinfo);

					ERRxwarning(0xC352, 2, "FileIO: Open Dir");

					/* Get FBK output information */
					fm->_numfiles	= fm->_dirinfo.filenum;
					fm->_infostatus	= fm->_dirinfo.status;

					/* Directory Info: Returned */
					if ( fm->_infostatus == 0 )	{
						fm->_fileptr	= 0;
						/* File Name Limit */
						if ( fm->_numfiles > fm->MaxDirectoryFiles )
							fm->_numfiles = fm->MaxDirectoryFiles;

						/* Init File Name Base Pointer */
						fname	= (fiDIR_READ_DATA *) fm->_fname_adr;

						ERRxwarning(0xC353, 3, "FileIO: Open Dir");
						ERRxwarning(0xC353, fm->_fname_adr, "FileIO: _fname_adr");

						/* Clear Array */
						for (i=0;i<fm->MaxDirectoryFiles;i++,fname++)
							memset( fname, 0, sizeof(fiDIR_READ_DATA) );

						/* Return File Names: */
						fm->_state++;

						/* Message */
						strcpy( fm->Message, "Reading Directory...Please Wait");
						ERRxwarning(0xC354, 4, "FileIO: Open Dir");
					}

					/* Directory Info: Unsuccessful */
					else if ( fm->_infostatus != 65535) {
						strcpy( fm->Message, "FileIO: Directory Info: Error");
						if ( fm->_infostatus == 20799)
							fm->Error = FileIoGetSysError();
						fm->_state 			= 100;
						fm->Status			= -1;				/* FileIO: Open Directory Error */
					}
				}
			}

			/* Method: Select Pattern: Process File */
			else if ( out->OpenFile | out->Save ) {

				/* Selected File has file name */
				if ( strcmp(out->SelectedFile, "") != 0) {

					/* Init File Name Base Pointer */
					fname	= (fiDIR_READ_DATA *) fm->_fname_adr;

					/* To Upper Case */
					ConvertToUpper( out->SelectedFile );

					/* Cycle Array: Directory */
					for (i=0;i<fm->MaxDirectoryFiles;i++,fname++) {

						/* Located File Index: */
						if ( strcmp( out->SelectedFile, fname->Filename) == 0 ) {
							FileFound	= 1;
							break;
						}
					}
				}

				/* Null Selected File: Error */
				else {
					strcpy( fm->Message, "FTP: Null File Name");
					out->OpenFile = 0;
				}

				if ( FileFound ) {

					/* Reset Status */
					fm->Status 			= 0;

					/* File Size Error: Streaming can have much larger file size than buffer */
					if ( (fname->Filelength > fm->BufferSize) && (fm->Type != FU_DRIVE_STREAM )) {
						strcpy( fm->Message, "File Open: Too Big");
						fm->_state			= 100;
						fm->Status			= -2;				/* File Open: File is too big */
					}

					/* File Size: Okay */
					else {

						/* FTP ...Talk to Goran
						if ( fm->Type == fuDRIVE_FTP ) {*/
						if ( fm->Type == 99 ) {

						}

						/* File IO */
						else {
							/* Initialize file open structrue */
							fm->_fileopen.pFile		= (UDINT) fname->Filename;

							/* Call FBK */
							FileOpen(&fm->_fileopen);

							/* Get FBK output information */
							fm->_fileopenstatus = fm->_fileopen.status;

							/* File Open: Doesn't Exist */
							if (fm->_fileopenstatus == 20708) {
								strcpy( fm->Message, "File Open: Does not Exist");
								fm->_state			= 100;
								fm->Status			= -3;				/* File Open: File does not exist */
							}

							/* File Open: Success */
							else if (fm->_fileopenstatus == 0) {
								/* Get Name */
								strcpy( fm->OpenFileName, fname->Filename  );
								fm->OpenFileDate	= fname->Date;
								strcpy( in->OpenFileName, fm->OpenFileName );
								GetExtType( in, out );
								/* Get Size */
								in->FileLength = fname->Filelength;
								/* Reset Status */
								fm->Status 			= 2;
								strcpy( fm->Message, "File Open: Success");

								/* Next Step */
								if ( out->OpenFile ) {
									fm->_fileread.pDest	= fm->Data_adr;
									memset( (void *) fm->_fileread.pDest, 0, fm->BufferSize );
									/* Streaming Read */
									if ( out->StreamEnable ) {
										fm->_state		= 10;
										fm->Status		= 10;
										out->OpenFile 	= 0;
									}
									/* Standard Read: Clear Memory */
									else	 {
										fm->_state		= 2;
									}
								}
								else if ( out->Save )
									fm->_state		= 3;	/* File Write */
							}

							/* File Open: File Not Found */
							else if ( fm->_fileopenstatus == fiERR_FILE_NOT_FOUND ) {
								strcpy( fm->Message, "File Open: Not Found");
								out->Save	= 0;
								fm->Status	= 10;				/* File Open: File does not exist */
							}

							/* File Open: Error */
							else if (fm->_fileopenstatus != 65535) {
								strcpy( fm->Message, "File Open: Error");
								fm->_state			= 100;
								fm->Status			= -4;				/* File Open: File Error */
								if (fm->_fileopenstatus == 20799)
									fm->Error = FileIoGetSysError();
							}
						}
					}
				}

				/* Can't Find File */
				else {
					strcpy( fm->Message, "Can not find file");
					out->Save	= 0;
					fm->Status	= -6;				/* File Open: File does not exist */
					fm->_state	= 100;
				}
			}

			/* NEW: Use out->SelectedFile */
			/* Delete File */
			else if ( out->DeleteFile ) {

				fm->Status	= 0;

				/* To Upper Case */
				ConvertToUpper( out->SelectedFile );

				/* Initialize file Delete structrue */
				fm->_filedelete.pName 	= (UDINT) out->SelectedFile;

				/* Call FBK */
            			FileDelete(&fm->_filedelete);

				/* Get FBK output information */
            			fm->_infostatus	= fm->_filedelete.status;

				/* Directory Info: Returned */
				if ( fm->_infostatus == 0 ) {
					strcpy( fm->Message, "Delete File: Success");
					out->DeleteFile 	= 0;
					fm->Status		= 1;
				}

				/* Delete Info: Not Found...still ok */
				else if ( fm->_infostatus == fiERR_FILE_NOT_FOUND ) {
					strcpy( fm->Message, "Delete File: File Not Found");
					out->DeleteFile 	= 0;
					fm->Status		= 1;
				}

				/* Directory Info: Unsuccessful */
				else if ( fm->_infostatus != 65535) {
					strcpy( fm->Message, "Delete File: Error!");
					out->DeleteFile 	= 0;
					fm->Status		= -1;
				}
			}

			/* Method: */
			else if ( out->CopyFile ) {

				if(!fm->Data_adr) return -100;

				/* Processing: */
				fm->Status		= 0;

				/* To Upper Case */
				ConvertToUpper( out->SelectedFile );

				/* Initialize file Copy structrue */
				fm->_filecopy.pSrc		= (UDINT) out->SelectedFile;
				fm->_filecopy.pDest		= 0;		/* Same Name */

				/* Call FBK */
				FileCopy(&fm->_filecopy);

				/* Copy File: Doesn't Exist */
				if (fm->_filecopy.status == 20708) {
					strcpy( fm->Message, "Copy File: Does not Exist");
					out->CopyFile 	= 0;
				}

				/* Copy File: Success */
				else if (fm->_filecopy.status == 0) {
					strcpy( fm->Message, "Copy File: Success");
					out->CopyFile 	= 0;
					fm->Status		= 4;
				}

				/* Copy File: Error */
				else if (fm->_filecopy.status != 65535) {
					strcpy( fm->Message, "Copy File: Error");
					out->CopyFile = 0;
				}
			}

			/* Method */
			else if ( out->SaveAs ) {

				/* Reset Status */
				fm->Status 			= 0;

				/* Create with Extension */
				if ( CreateNewFileName(out) == 0 ) {

					/* Initialize file create structrue */
					fm->_filecreate.pFile	= (UDINT) out->SelectedFile;

					/* Call FBK */
					FileCreate(&fm->_filecreate);

					/* Get FBK output information */
					fm->_filecreatestatus = fm->_filecreate.status;

					/* No Need To Go to Error State! */
					/* File Already Exists: 20705 */
					if (fm->_filecreatestatus == fiERR_EXIST ) {
						strcpy( fm->Message, "File Exists: Updating..");
						out->SaveAs 	= 0;
						out->Save		= 1;
						fm->_state		= 0;
					}

					/* File Create: Success */
					else if (fm->_filecreatestatus == 0) {
						strcpy( fm->Message, "File Create: Success");
						fm->Status		= 3;
						fm->_state		= 3;	/* File Create Success: Perform File Write */
					}

					/* File Create: Error */
					else if (fm->_filecreatestatus != 65535) {
						strcpy( fm->Message, "File Create: Error");
						fm->_state		= 100;
						fm->Status		= -5;				/* File Create: Error */
						if (fm->_filecreatestatus == fiERR_SYSTEM)
							fm->Error = FileIoGetSysError();
					}
				}
				else {
					strcpy( fm->Message, "File Create: Bad Extension");
					fm->Status		= -6;				/* File Create: Bad Extension */
					fm->_state		= 100;
				}
			}

		break;

		/**** Return File Names ****/
		case 1:

			/* Read File Names */
			if (fm->_fileptr < fm->_numfiles) {

				/* Init: Dynamic Read Info */
				fm->_dirread.entry 		= fm->_fileptr;

				/* Init File Name Base Pointer: Then Index */
				fname	= (fiDIR_READ_DATA *) fm->_fname_adr;
				fname 	+= fm->_fileptr;

				/* Initialize Directory Read structrue */
				fm->_dirread.pData 		= (UDINT) fname->Filename;

				/* Call FBK */
				DirRead(&fm->_dirread);

				/* Update Read Status */
				fm->_readstatus		= fm->_dirread.status;

				/* Directory Read: Returned */
				if ( fm->_readstatus == 0) {
					ConvertToUpper( fname->Filename );
					strcpy( fm->Message, "Directory Read: OK");
					fm->_fileptr++;
				}

				/* Directory Read: Unsuccessful */
				else if (fm->_readstatus != 65535)	{
					fm->Status		= -7;				/* Directory Read Error */
					fm->_state 		= 100;
					strcpy( fm->Message, "Directory Read: Error");
					if ( fm->_readstatus == 20799)
						fm->Error = FileIoGetSysError();
				}
			}

			/* File Names Read */
			else {
				strcpy( fm->Message, "Directory Read: Completed");
				fm->_state			= 0;
				fm->Status 			= 1;
				out->OpenDirectory	= 0;
				FilterExt			= 1;
			}

		break;

		/**** Read data from file ****/
		case 2:

			/* Initialize file read structure */
			fm->_fileread.ident 	= fm->_fileopen.ident;
			fm->_fileread.pDest	= fm->Data_adr;

			/* Call FBK */
			FileRead(&fm->_fileread);

			/* Get status */
			fm->_filereadstatus = fm->_fileread.status;

			/* File Read: Success */
			if (fm->_filereadstatus == 0) {
				fm->_state 			= 4;
				out->OpenFile 		= 0;
				fm->_fileclose.ident = fm->_fileread.ident;
				strcpy( fm->Message, "File Read: Success");
			}
			/* File Read: Error */
			else if (fm->_filereadstatus != 65535)	{
				strcpy( fm->Message, "File Read: Error");
				out->OpenFile 		= 0;
				fm->_state 			= 101;
				fm->Status			= -9;				/* File Read Error */
				fm->_fileclose.ident = fm->_fileread.ident;
				if (fm->_filereadstatus == 20799)
					fm->Error = FileIoGetSysError();
			}

		break;

		/**** File Write: Part 2 of out->SaveAs Method ****/
		case 3:

			/* Initialize file write structure */
			if ( out->SaveAs )
				fm->_filewrite.ident 	= fm->_filecreate.ident;
			else if ( out->Save )
				fm->_filewrite.ident	= fm->_fileopen.ident;

			/* Size */
			fm->_filewrite.len 			= out->FileSize;
			fm->_filewrite.pSrc		= fm->Data_adr;

			/* Clear Commands */
			out->SaveAs	= 0;
			out->Save   = 0;

			/* Call FBK */
			FileWrite(&fm->_filewrite);

			/* Get status */
			fm->_filewritestatus = fm->_filewrite.status;

			/* File Write: Success */
			if (fm->_filewritestatus == 0) {
				fm->_state 	= 4;
				fm->_fileclose.ident = fm->_filewrite.ident;
				strcpy( fm->Message, "File Write: Success");
			}
			/* File Write: Error */
			else if (fm->_filewritestatus != 65535)	{
				strcpy( fm->Message, "File Write: Error");
				fm->Status	= -10;				/* File Write Error */
				fm->_state 	= 101;
				fm->_fileclose.ident = fm->_filewrite.ident;
				if (fm->_filewritestatus == 20799)
					fm->Error = FileIoGetSysError();
			}

		break;

		/**** FileClose: called after each fileRead or fileWrite ****/
		case 4:

			/* Call FBK */
			FileClose(&fm->_fileclose);

			/* Verify status */
			if (fm->_fileclose.status == 0)  {
				fm->Status	= 4;
				fm->_state	= 0;
			}
			else if (fm->_fileclose.status != 65535) {
				strcpy( fm->Message, "File Close: Error");
				fm->Status	= -11;				/* File Close Error */
				fm->_state 	= 0;
				if (fm->_fileclose.status == 20799)
		 			fm->Error = FileIoGetSysError();
			}

		break;

		/********************************************************************/
		/**** Streaming Output ****/
		case 10:

			/* Wait Stream Command: Initialize file read structure */
			if ( out->StreamGo ) {
				fm->_fileread.ident 	= fm->_fileopen.ident;
				fm->_fileread.offset	= out->StreamOffset;
				fm->_fileread.len		= out->StreamLength;
				fm->_fileread.pDest	= out->Stream_adr;
				/* Response Signals: Reset */
				in->StreamReady		= 0;
				in->StreamError		= 0;
				fm->_state++;
			}

			/* Close Connection */
			else if ( out->StreamClose ) {
				out->StreamClose		= 0;
				fm->_fileclose.ident 	= fm->_fileread.ident;
				fm->_state			= 4;
			}

		break;

		/********************************************************************/
		/**** Streaming Output ****/
		case 11:

			/* Call FBK */
			FileRead(&fm->_fileread);

			/* Get status */
			fm->_filereadstatus = fm->_fileread.status;

			/* File Read: Success */
			if (fm->_filereadstatus == 0) {
				out->StreamGo		= 0;
				in->StreamReady		= 1;					/* Response: Ok */
				fm->_state 			= 10;
			}
			/* File Read: Error */
			else if (fm->_filereadstatus != 65535)	{
				out->StreamGo		= 0;
				in->StreamError		= 1;					/* Response: Error */
				fm->_state 			= 101;
				strcpy( fm->Message, "File Stream: Error");
				fm->Status			= -11;				/* File Stream: Error */
				fm->_fileclose.ident = fm->_fileread.ident;
				if (fm->_filereadstatus == 20799)
					fm->Error = FileIoGetSysError();
			}

		break;
		/********************************************************************/

		/**** Error State ****/
		case 100:

			/* Clear Commands */
			out->OpenDirectory 	= 0;
			out->OpenFile 		= 0;
			out->SaveAs 			= 0;
			out->Save			= 0;
			out->StreamClose		= 0;

			/* Command: Reset Error */
			fm->_state			= 0;

		break;

		/**** Error State w. FileClose ****/
		case 101:

			/* Call FBK */
			FileClose(&fm->_fileclose);

			/* Verify status */
			if (fm->_fileclose.status == 0)  {
				fm->_state	= 100;
			}
			else if (fm->_fileclose.status != 65535) {
				strcpy( fm->Message, "File Close: Error");
				fm->Status	= -12;				/* File Close Error */
				fm->_state 	= 100;
				if (fm->_fileclose.status == 20799)
		 			fm->Error = FileIoGetSysError();
			}
		break;

		default:
		break;

	}

	/* Input Interface: Files in Directory */
	in->TotalDirectoryFileNum	= fm->_numfiles;
	/* Input Interface: Message */
	strcpy( in->Message, fm->Message );

	/* Process Page Scroll: Up */
	if ( out->PageUp ) {
		out->PageUp = 0;
		FilterExt 	= 1;
		if (in->PageNum > 0)
			in->PageNum--;
	}
	/* Process Page Scroll: Down */
	if ( out->PageDown ) {
		out->PageDown 	= 0;
		FilterExt		= 1;
		if (in->PageNum < (FU_MAX_PAGE_FILES-1) && (in->TotalPageFileNum == FU_MAX_PAGE_FILES) )
			in->PageNum++;
	}

	/* Perform Extension Filter */
	if ( FilterExt | out->Refresh ) {

		/* Reset */
		out->Refresh	= 0;

		/* Locate Total Files per Extension */
		j = 0;

		/* Init File Name Base Pointer */
		fname	= (fiDIR_READ_DATA *) fm->_fname_adr;

		/* Cycle Array */
		for (i=0;i<fm->_numfiles;i++,fname++) {

			/* All Extensions */
			if ( out->ExtensionIndex == 0 )
				j++;

			/* Special: Extension 0 and 1: Specific Extension */
			else if ( out->ExtensionIndex == 10 ) {
				if (	(FindString( fname->Filename, out->Extension[0].Name) == 0) ||
					(FindString( fname->Filename, out->Extension[1].Name) == 0) )
					j++;
			}

			/* Specific Extension */
			else if ( out->ExtensionIndex <= FU_MAX_EXT ) {
				if (FindString( fname->Filename, out->Extension[out->ExtensionIndex-1].Name) == 0 )
					j++;
			}
		}

		/* Assign */
		in->TotalDirectoryFileNum	= j;

		/* Locate Total Page Files per Extension */
		j = 0;

		/* Page Scroll Index */
	    StartIndex = in->PageNum * FU_MAX_PAGE_FILES;

		/* Clear */
		for (i=0;i<FU_MAX_PAGE_FILES;i++) {
			memset( (UDINT *) &in->FileNames[i][0], 0, sizeof(in->FileNames[0]));
			in->FileDates[i] = 0;
			in->FileSizes[i] = 0;
		}

		/* Init File Name Base Pointer */
		fname	= (fiDIR_READ_DATA *) fm->_fname_adr;

		/* Cycle Array */
		for (i=0;i<fm->_numfiles;i++,fname++) {

			/* View All Extensions */
			if ( out->ExtensionIndex == 0 ) {
				if ( j >= StartIndex ) {
					strcpy( &in->FileNames[j-StartIndex][0], fname->Filename );
					in->FileDates[j-StartIndex]	= fname->Date;
					in->FileSizes[j-StartIndex]	= fname->Filelength;
				}
				j++;
			}

			/* Special: Allow Index 0 and 1 */
			else if ( out->ExtensionIndex == 10 ) {
				if ( 	(FindString( fname->Filename, out->Extension[0].Name) == 0) ||
					(FindString( fname->Filename, out->Extension[1].Name) == 0) ) {
					if ( j >= StartIndex ) {
						strcpy( &in->FileNames[j-StartIndex][0],fname->Filename);
						in->FileDates[j-StartIndex]	= fname->Date;
						in->FileSizes[j-StartIndex]	= fname->Filelength;
					}
					j++;
				}
			}

			/* Locate File with Proper Extension */
			else if ( out->ExtensionIndex <= FU_MAX_EXT ) {
				if (FindString( fname->Filename, out->Extension[out->ExtensionIndex-1].Name) == 0 ) {
					if ( j >= StartIndex ) {
						strcpy( &in->FileNames[j-StartIndex][0],fname->Filename);
						in->FileDates[j-StartIndex]	= fname->Date;
						in->FileSizes[j-StartIndex]	= fname->Filelength;
					}
					j++;
				}
			}

			/* Check Page Disply Limit */
			if ( j >= (StartIndex + FU_MAX_PAGE_FILES) ) {
				break;
			}

		}

		/* Files in Page View */
		in->TotalPageFileNum 		= j - StartIndex;
	}

	/* Method: Clear Status */
	if ( out->ClearStatus )  {
		out->ClearStatus 	= 0;
		fm->Status			= 0;
	}
	in->Status				= fm->Status;

	return 0;
}
/*********************************************************
* NAME		:	FU_AddExt (Public)
*
* OBJECT	:	FILEOUT_IF, FILEIN_IF
*
* FUNCTION	:	Changes the OpenFileName string to the supplied
				extension index

				i.e.	.OpenFileName	= "PatternFile1.ctf"
					.ExtensionIndex	= 2 	("col")

					Result:

					.OpenFileName	= "PatternFile1.col"
*
*
* PARAMETERS:	out
				in

*
* RETURN	:	-1: 		Error "." not found
				0:		Success
				1:		Bad Extension Index
*
* HISTORY	:	02.07.07 - Version 1

*********************************************************/
DINT FU_AddExt( FILEOUT_IF *out, FILEIN_IF *in )
{
STRING base[34];
USINT i;

	/* Get Local Copy */
	strcpy( base, in->OpenFileName );

	/* Locate '.' */
	for (i=0;i<strlen(base);i++) {
		if ( base[i] == '.' ) {
			base[i] = 0;			/* Add Null */
			strcpy( out->NewFileNameBase, base	);
			return CreateNewFileName( out );
		}
	}

	return -1;
}

 /* */
BOOL FU_DeleteExt( STRING s[35], STRING d[35])
{
USINT i;

	/* Locate '.' */
	for (i=0;i<strlen(s);i++) {
		d[i]	= s[i];
		if ( s[i] == '.' ) {
			d[i]	= 0;
			return 1;
		}
	}

	/* Not Found */
	return 0;
}

#if 0
DINT FU_AddExt( UDINT fm_adr, STRING s[35], STRING ext[4] )
{
FILEMGR_obj *fm	= (FILEMGR_obj *) fm_adr;
FILEOUT_IF *out	= (FILEOUT_IF  *) fm->_if_out_adr;
STRING _s[35];
USINT i;

	/* Source String: Local Copy */
	strcpy( _s, s );

	/* Locate '.' */
	for (i=0;i<strlen(_s);i++) {
		/* Found Extension */
		if ( _s[i] == '.' ) {
			memcpy( &_s[i+1], ext, 3);
			/* Add Null */
			_s[i+4] = 0;
			/* To Upper */
			ConvertToUpper( _s );
			/* Copy */
			strcpy( out->SelectedFile, _s );
			/* Return */
			return (i);
		}
	}

	return 0;
}
#endif

void ConvertToUpper( STRING s[35] )
{
UINT i;

	/* Verify Letters Only */
	for (i=0;(i<strlen(s)) && (i<35);i++) {
		if ( ((s[i] >= 'A') && (s[i] <= 'Z')) ||
			 ((s[i] >= 'a') && (s[i] <= 'z'))    ) {
			s[i] = s[i] & 0xDF;
		}
	}
}

/* */
DINT FindString( STRING s[35], STRING ext[4] )
{
USINT i, j, s_ext[5];

	/* Locate '.' */
	for (i=0;i<strlen(s);i++) {
		if ( s[i] == '.' ) {
			/* Convert to Next 3 Chars to Upper */
			for (j=1;j<4;j++)
				s[i+j] = s[i+j] & 0xDF;
			memcpy( s_ext,&s[i], 4);
			/* Add Null */
			s_ext[4] = 0;
			return strcmp(s_ext, ext);
			break;
		}
	}

	/* Not Found */
	return 255;
}

/* */
DINT GetExtType( FILEIN_IF *in, FILEOUT_IF *out )
{
USINT i,j, s_ext[5];

	/* Locate '.' */
	for (i=0;i<strlen(in->OpenFileName);i++) {
		if ( in->OpenFileName[i] == '.' ) {
			memcpy( s_ext,&in->OpenFileName[i], 4);
			/* Add Null */
			s_ext[4] = 0;
			for (j=0;j<5;j++) {
				if (strcmp(s_ext, out->Extension[j].Name) == 0) {
					in->ExtensionIndex = j;
					return 0;
				}
			}
		}
	}

	/* */
	return -1;
}

DINT CreateNewFileName( FILEOUT_IF *out )
{
STRING base[34];

	if ( (FU_MAX_EXT + 1) > out->ExtensionIndex > 0 ) {
		/* Process */
		memset( base, 0, sizeof(base));
		strcpy( base, out->NewFileNameBase );
		strcat( base, out->Extension[out->ExtensionIndex-1].Name );
		strcpy( out->SelectedFile, base);
		return 0;
	}
	else
		return 1;
}

UINT SortDirectory( UDINT fm_adr )
{
FILEMGR_obj *fm			= (FILEMGR_obj *) fm_adr;
fiDIR_READ_DATA *s1, *s2;
fiDIR_READ_DATA hold;
UINT i,j=0;

	/* Init File Name Base Pointer */
	s1	= (fiDIR_READ_DATA *) fm->_fname_adr;
	s2	= (fiDIR_READ_DATA *) fm->_fname_adr;

	s2++;

		/* Cycle Array: Compare */
		for (i=1;i<fm->_numfiles;i++,s1++,s2++) {
			if ( strcmp(s1->Filename, s2->Filename) > 0 ) {
				memcpy( &hold, s1, 	sizeof(fiDIR_READ_DATA));
				memcpy( s1, s2, 		sizeof(fiDIR_READ_DATA));
				memcpy( s2, &hold, 	sizeof(fiDIR_READ_DATA));
				j++;
			}
		}

	return j;
}
```

#### FU_setMem.c
```c
/********************************************************************
 * COPYRIGHT --
 ********************************************************************
 * Library: FileUser
 * File: FU_setMem.c
 * Author: ChrisK
 * Created: October 22, 2009
 ********************************************************************
 * Implementation of library FileUser
 ********************************************************************/

#include <bur/plctypes.h>
#include "FileUser.h"

/*TODO: Add your comment here*/
plcbit FU_setMem(unsigned long pMem, unsigned long size)
{
	/*TODO: Add your code here*/
}
```

### Library Logical/Libraries/XMLp_Lib (ANSIC, version 1.54.0)
Depends on: SYS_LIB, AsString

#### XMLp_Lib.fun
```iecst
FUNCTION XMLp_CallParse : DINT
	VAR_INPUT
		m : XML_Method_typ;
	END_VAR
END_FUNCTION

FUNCTION XMLp_CallCreate : DINT
	VAR_INPUT
		m : XML_Method_typ;
		PVNames : REFERENCE TO USINT;
	END_VAR
END_FUNCTION

FUNCTION XMLp_Init : BOOL
	VAR_INPUT
		m : XML_Method_typ;
		BufferSize : UDINT;
	END_VAR
END_FUNCTION

FUNCTION XMLp_Destroy : BOOL (*TODO: Add your comment here*)
	VAR_INPUT
		m : XML_Method_typ;
	END_VAR
END_FUNCTION
```

#### XMLp_Lib.typ
```iecst
TYPE
	XML_ParseInfo_typ : 	STRUCT
		LinesProcessed : UINT;
		LengthInBytes : UDINT;
		ErrorNum : DINT;
		ItemsNotFound : UINT;
		ErrorMessage : ARRAY[0..9] OF STRING[50];
		IgnoreNotFound : BOOL;
	END_STRUCT;
	XML_CreateInfo_typ : 	STRUCT
		LengthInBytes : UDINT;
		ErrorNum : DINT;
	END_STRUCT;
	XML_DiagInfo_typ : 	STRUCT
		Reset : BOOL;
		Logger : BOOL;
		TotalCalls : UDINT;
		TotalResponses : UDINT;
		TotalFaults : UDINT;
		TotalErrors : UDINT;
	END_STRUCT;
	XML_Method_typ : 	STRUCT
		InitStatus : DINT;
		Status : DINT;
		MethodName : STRING[40];
		PVServer : STRING[40];
		PVClient : STRING[40];
		OpIndex : INT;
		ParseInfo : XML_ParseInfo_typ;
		CreateInfo : XML_CreateInfo_typ;
		DiagInfo : XML_DiagInfo_typ;
		Fault : BOOL;
		FaultString : STRING[40];
		FaultCode : DINT;
		ViewLineString : STRING[119];
		ViewInc : BOOL;
		ViewLine : UINT;
		ViewLevel : UINT;
		_viewline : UINT;
		BufferSize : UDINT;
		pMessage : UDINT;
	END_STRUCT;
END_TYPE
```

#### XMLp_Lib.var
```iecst
VAR CONSTANT
	XMLp_STATUS_SUCCESS	: SINT	:= 5;
	XMLp_STATUS_FAULT	: SINT	:= 3;
END_VAR
```

#### xml_def.h
```c
/*********************************************************
* FILE		:		xml_def.h(Header)
*
* OBJECTs	:
*
* OVERVIEW	:
*
*
* HISTORY : 			08.31.07	- Version 1.0
					09.18.07	- Version 1.1
					02.14.08	- STRING_LENGTH_MAX 40
					02.28.08	- STRING Null

*
* DEPENDANCIES:
*********************************************************/
#include <bur/plc.h>
#include <bur/plctypes.h>
#include <xmlp_lib.h>

/* DEFINES:
*********************************************************/
#ifndef OFF
	#define OFF 0
	#define ON 1
	#define YES 1
	#define NO 0
#endif
#ifndef STRING_LENGTH_MAX
	#define STRING_LENGTH_MAX			40
#endif

/* MACROS:
*********************************************************/
#define XML_BODY_VERSION				"<?xml version=\"1.0\" encoding=\"utf-8\"?>"
#define XML_BODY_OPEN					"<"
#define XML_BODY_CLOSE					"</"
#define XML_BODY_END					">"

#define XML_BODY_METHOD_CALL			"methodCall"
#define XML_BODY_METHOD_RESPONSE		"methodResponse"
#define XML_BODY_METHOD_NAME			"methodName"
#define XML_BODY_PARAMS					"variables"
#define XML_BODY_PARAM					"variable"
#define XML_BODY_VALUE					"value"
#define XML_BODY_STRUCT				"struct"
#define XML_BODY_ARRAY					"array"
#define XML_BODY_DATA					"data"
#define XML_BODY_MEMBER 				"member"
#define XML_BODY_NAME					"name"
#define XML_BODY_FAULT					"fault"
#define XML_BODY_FAULT_CODE			"faultCode"
#define XML_BODY_FAULT_STRING 		"faultString"

#define XML_BODY_TYPE_I4				"i4"
#define XML_BODY_TYPE_I4_V1			"integer"			/* Variant */
#define XML_BODY_TYPE_BOOL			"boolean"
#define XML_BODY_TYPE_STRING			"string"
#define XML_BODY_TYPE_DOUBLE			"double"
#define XML_BODY_TYPE_DATE_TIME			"date_time"			//"dateTime.iso8601"

#define XML_OP_READ					"Read"
#define XML_OP_READ_2 					"read"
#define XML_OP_READ_3 					"READ"
#define XML_OP_READ_IDX				1
#define XML_OP_WRITE 					"Write"
#define XML_OP_WRITE_2					"write"
#define XML_OP_WRITE_3					"WRITE"
#define XML_OP_WRITE_IDX 				2
#define XML_OP_METHOD					"Method"
#define XML_OP_METHOD_2				"method"
#define XML_OP_METHOD_3 				"METHOD"
#define XML_OP_METHOD_IDX 				3
#define XML_OP_FILEWRITE				"FileWrite"
#define XML_OP_FILEWRITE_IDX			12
#define XML_OP_FILEREAD				"FileRead"
#define XML_OP_FILEREAD_IDX			13

#define XML_CLOSE							1
#define XML_OPEN							0

#define XML_BODY_TYPE_NULL_IDX			0
#define XML_BODY_TYPE_I4_IDX				1
#define XML_BODY_TYPE_BOOL_IDX			2
#define XML_BODY_TYPE_STRING_IDX			3
#define XML_BODY_TYPE_DOUBLE_IDX			4
#define XML_BODY_TYPE_DATE_TIME_IDX			5

#define XML_BODY_PARAM_IDX				30
#define XML_BODY_PARAMS_IDX				31
#define XML_BODY_METHOD_CALL_IDX			32
#define XML_BODY_STRUCT_IDX				33
#define XML_BODY_VALUE_IDX					34
#define XML_BODY_METHOD_RESPONSE_IDX	35
#define XML_BODY_FAULT_IDX					36
#define XML_BODY_MEMBER_IDX				37
#define XML_BODY_METHOD_NAME_IDX			38
#define XML_BODY_NAME_IDX					39
#define XML_BODY_ARRAY_IDX				40
#define XML_BODY_DATA_IDX					41

#define XML_BODY_INDENT_1					"	"

#define XML_VERSION 						999

#ifndef TYPE_BOOL
	#define TYPE_BOOL						1
	#define TYPE_SINT						2
	#define TYPE_INT						3
	#define TYPE_DINT						4
	#define TYPE_USINT						5
	#define TYPE_UINT						6
	#define TYPE_UDINT						7
	#define TYPE_REAL						8
	#define TYPE_STRING						9
	#define TYPE_DATE_TIME					11
	#define TYPE_TIME						12
#endif

#define cTAB		9
#define cLF		10
#define cCR 		13
#define cSLASH	47
#define cLT		60
#define cGT		62
#define cQUESTION	63

#define LINE_LENGTH_MAX			120
#define XML_CLIENT					"client"
#define XML_SERVER					"server"
#define XML_FAULT_CODE				"fault.Code"
#define XML_FAULT_STRING			"fault.String"
#define XML_TRUE					"true"
#define XML_FALSE					"false"
#define XML_STRING_NULL			"NULL"

/* Client Status */
#define XMLd_STATUS_ERROR			-100
#define XML_STATUS_RESP_ERROR		-2
#define XML_STATUS_CALL_ERROR		-1
#define XML_STATUS_READY			0
#define XML_STATUS_SENDNOW		1
#define XML_STATUS_METHOD			2
#define XML_STATUS_FAULT 			3
#define XML_STATUS_FAULT_AUTO		4
#define XML_STATUS_COMPLETE		5
#define XML_STATUS_PARSE_OK	 	6

#define XML_BUFFER_REMAIN			500

/* TYPES:
*********************************************************/
typedef struct {
	STRING 	Name[STRING_LENGTH_MAX];
	UDINT	Length;
	UDINT	Type;
	UINT	Dim;
} DataElement_typ;

typedef struct {
	DINT	Key[4];

	UINT	NumKeys;
	UINT	NumOpenKeys;
	UINT	NumCloseKeys;
	UINT	NumValues;
	STRING	sValue[STRING_LENGTH_MAX];
	REAL	rValue;
	DINT	iValue;
	BOOL	bValue;
} LineElement_typ;

/* HELPER PROTOTYPES:
*********************************************************/
DINT xml_FaultDetected( XML_Method_typ *m,	DINT FaultCode, STRING FaultString[STRING_LENGTH_MAX], UDINT offset );
DINT xml_FaultDetectedInResponse( XML_Method_typ *m,	DINT FaultCode, STRING FaultString[STRING_LENGTH_MAX] );
BOOL xml_MessageViewer( XML_Method_typ *m, UINT line, USINT *text );
DINT xml_AddItems( USINT *msg, char* PVBaseName, UINT *Indent, UDINT	*offset, UDINT BufferSize, BOOL Logger );
DINT xml_AppendIndex( STRING Dest[100], USINT num );
DINT xml_GetLineInformation( XML_Method_typ *m, UDINT	*offset, LineElement_typ *line, BOOL *lastlinedected );
DINT xml_GetElement( XML_Method_typ *m, STRING *pBaseName, UDINT	*offset, UINT idx, LineElement_typ *line);
DINT xml_ProcessValue( STRING *pName, LineElement_typ *line, UINT idx );
DINT xml_SetErrorFlag( XML_Method_typ *m  );
DINT xml_CreateFaultMessage( XML_Method_typ *m,  UDINT	*offset, DINT FaultCode, STRING FaultString[STRING_LENGTH_MAX] );
DINT xml_InsertComplexLine( USINT *msg, UINT Type, UINT size, UDINT  *offset, void *pData, UINT Indent);
DINT xml_InsertKey( USINT *msg, UINT Type, UDINT  *offset, UINT Indent, BOOL Option );
DINT xml_GetKeyIndex( USINT *pItemText, BOOL *SlashFound );
DINT xml_GetOpIndex( USINT *pOpName );
UINT xml_DataTypeToValueType(  UDINT type );
DINT xml_MakeCallName(	USINT *pDest, USINT *pOpName, USINT *pMethodName );
DINT _xmlGetStringFromFile( USINT *f0, UDINT  *offset, USINT *dest );
DINT _xmlGetLine( USINT *f0, UDINT	*offset, USINT *dest, BOOL *lastline, UINT *levels );
BOOL _GetStringFromFile( USINT *f0, UDINT  *offset, USINT *dest, USINT *endchar, BOOL ignore );
void _AddIntToFile( USINT *f0, UDINT  *offset, INT x, USINT *endchar );
void _AddDintToFile( USINT *f0, UDINT  *offset, DINT x, USINT *endchar );
void _AddFloatToFile( USINT *f0, UDINT	*offset, REAL x, USINT *endchar );
void _AddStringToFile( USINT *f0, UDINT  *offset, USINT *s, USINT *endchar );
signed long AddIndex(plcstring* Dest, plcstring* Name, unsigned char num);
/* EOF */
```
